// TwinCAT 3 PLC project AssemblyDemo
// ProgramVersion: 3.1.4024.0
// libraries:
//   Tc3_Module, * (Beckhoff Automation GmbH)
//   ZApplication, 1.5.8.2 (Zeugwerk GmbH)
//   ZAux, 1.5.8.2 (Zeugwerk GmbH)
//   ZCore, 1.5.8.2 (Zeugwerk GmbH)
//   ZEquipment, 1.5.8.2 (Zeugwerk GmbH)
//   ZPlatform, 1.5.8.2 (Zeugwerk GmbH)
// project tree:
//   ZApp/App/ ZApp.TcPOU
//   ZApp/App/_DataTypes/ ZAppStep.TcDUT
//   ZApp/App/_States/ ZAppSequenceBoot.TcPOU, ZAppSequenceBootFault.TcPOU, ZAppSequenceRunning.TcPOU
//   ZApp/App/_SubObjects/ ZAppSequence.TcPOU
//   ZApp/Com/_DataTypes/ ZCom.TcDUT, ZComUnit.TcDUT
//   ZApp/Data/_DataTypes/ ZData.TcDUT, ZDataMachine.TcDUT, ZDataConfig.TcDUT, ZDataCalibration.TcDUT, ZDataRecipe.TcDUT
//   ZApp/Unit/Assembly/ AssemblyUnit.TcPOU, AssemblyUnitProgram.TcPOU, IAssembly.TcIO
//   ZApp/Unit/Assembly/_Com/ AssemblyCom.TcDUT, AssemblyComPublish.TcDUT, AssemblyComPublishEquipment.TcDUT, AssemblyComRef.TcDUT, AssemblyComRequest.TcDUT, AssemblyComSubscribe.TcDUT, AssemblyComSubscribeEquipment.TcDUT
//   ZApp/Unit/Assembly/_DataTypes/ ActuatorHorizontalListenerStep.TcDUT, AssemblyState.TcDUT, AssemblyStep.TcDUT
//   ZApp/Unit/Assembly/_Data/ AssemblyDataCalibration.TcDUT, AssemblyDataConfig.TcDUT, AssemblyDataMachine.TcDUT, AssemblyDataRef.TcDUT
//   ZApp/Unit/Assembly/_Equipment/ ActuatorHorizontalListener.TcPOU, AssemblyActuator.TcPOU, AssemblyActuatorGripper.TcPOU, AssemblyActuatorHorizontal.TcPOU, AssemblyAxis.TcPOU, AssemblyEquipment.TcPOU, AssemblyFieldbus.TcPOU, AssemblyIo.TcPOU, AssemblyLinkedUnit.TcPOU, PneumaticsOkActuatorListener.TcPOU
//   ZApp/Unit/Assembly/_States/ AssemblySequenceAutomatic.TcPOU, AssemblySequenceBoot.TcPOU, AssemblySequenceFaultReaction.TcPOU, AssemblySequenceGoHome.TcPOU, AssemblySequenceStop.TcPOU
//   ZApp/Unit/Assembly/_SubObjects/ AssemblyContainer.TcPOU, AssemblySequence.TcPOU
//   ZApp/Unit/Drilling/ DrillingUnit.TcPOU, DrillingUnitProgram.TcPOU, IDrilling.TcIO
//   ZApp/Unit/Drilling/_Com/ DrillingCom.TcDUT, DrillingComPublish.TcDUT, DrillingComPublishEquipment.TcDUT, DrillingComRef.TcDUT, DrillingComRequest.TcDUT, DrillingComSubscribe.TcDUT, DrillingComSubscribeEquipment.TcDUT
//   ZApp/Unit/Drilling/_DataTypes/ DrillingState.TcDUT, DrillingStep.TcDUT
//   ZApp/Unit/Drilling/_Data/ DrillingDataCalibration.TcDUT, DrillingDataConfig.TcDUT, DrillingDataMachine.TcDUT, DrillingDataRef.TcDUT
//   ZApp/Unit/Drilling/_Equipment/ DrillingActuator.TcPOU, DrillingActuatorVertical.TcPOU, DrillingAxis.TcPOU, DrillingEquipment.TcPOU, DrillingFieldbus.TcPOU, DrillingIo.TcPOU, DrillingLinkedUnit.TcPOU
//   ZApp/Unit/Drilling/_States/ DrillingSequenceAutomatic.TcPOU, DrillingSequenceBoot.TcPOU, DrillingSequenceFaultReaction.TcPOU, DrillingSequenceGoHome.TcPOU, DrillingSequenceStop.TcPOU
//   ZApp/Unit/Drilling/_SubObjects/ DrillingContainer.TcPOU, DrillingSequence.TcPOU
//   ZApp/Unit/QualityInspection/ IQualityInspection.TcIO, QualityInspectionUnit.TcPOU, QualityInspectionUnitProgram.TcPOU
//   ZApp/Unit/QualityInspection/_Com/ QualityInspectionCom.TcDUT, QualityInspectionComPublish.TcDUT, QualityInspectionComPublishEquipment.TcDUT, QualityInspectionComRef.TcDUT, QualityInspectionComRequest.TcDUT, QualityInspectionComSubscribe.TcDUT, QualityInspectionComSubscribeEquipment.TcDUT
//   ZApp/Unit/QualityInspection/_DataTypes/ QualityInspectionState.TcDUT, QualityInspectionStep.TcDUT
//   ZApp/Unit/QualityInspection/_Data/ QualityInspectionDataCalibration.TcDUT, QualityInspectionDataConfig.TcDUT, QualityInspectionDataMachine.TcDUT, QualityInspectionDataRef.TcDUT
//   ZApp/Unit/QualityInspection/_Equipment/ QualityInspectionActuator.TcPOU, QualityInspectionAxis.TcPOU, QualityInspectionEquipment.TcPOU, QualityInspectionFieldbus.TcPOU, QualityInspectionIo.TcPOU, QualityInspectionLinkedUnit.TcPOU
//   ZApp/Unit/QualityInspection/_States/ QualityInspectionSequenceAutomatic.TcPOU, QualityInspectionSequenceBoot.TcPOU, QualityInspectionSequenceFaultReaction.TcPOU, QualityInspectionSequenceGoHome.TcPOU, QualityInspectionSequenceStop.TcPOU
//   ZApp/Unit/QualityInspection/_SubObjects/ QualityInspectionContainer.TcPOU, QualityInspectionSequence.TcPOU
//   ZApp/Unit/Transport/ ITransport.TcIO, TransportUnit.TcPOU, TransportUnitProgram.TcPOU
//   ZApp/Unit/Transport/_Com/ TransportCom.TcDUT, TransportComPublish.TcDUT, TransportComPublishEquipment.TcDUT, TransportComRef.TcDUT, TransportComRequest.TcDUT, TransportComSubscribe.TcDUT, TransportComSubscribeEquipment.TcDUT
//   ZApp/Unit/Transport/_DataTypes/ TransportState.TcDUT, TransportStep.TcDUT
//   ZApp/Unit/Transport/_Data/ TransportDataCalibration.TcDUT, TransportDataConfig.TcDUT, TransportDataMachine.TcDUT, TransportDataRef.TcDUT
//   ZApp/Unit/Transport/_Equipment/ TransportActuator.TcPOU, TransportActuatorGripper.TcPOU, TransportAxis.TcPOU, TransportEquipment.TcPOU, TransportFieldbus.TcPOU, TransportIo.TcPOU, TransportLinkedUnit.TcPOU
//   ZApp/Unit/Transport/_States/ TransportSequenceAutomatic.TcPOU, TransportSequenceBoot.TcPOU, TransportSequenceFaultReaction.TcPOU, TransportSequenceGoHome.TcPOU, TransportSequenceStop.TcPOU
//   ZApp/Unit/Transport/_SubObjects/ TransportContainer.TcPOU, TransportSequence.TcPOU
//   ZApp/ ZGlobal.TcGVL, ZModuleProgram.TcPOU, ZModuleTask.TcTTO
// real-time tasks:
//   TASK ZModuleTask: cycle T#10ms, priority 20, ADS port 350

CONFIGURATION AssemblyDemo
    RESOURCE PLC ON TwinCAT3
        TASK ZModuleTask(INTERVAL := T#10ms, PRIORITY := 20);
        PROGRAM ZModuleProgram WITH ZModuleTask : ZModuleProgram;
    END_RESOURCE
END_CONFIGURATION

// ---- ZApp/App/_DataTypes/ZAppStep.TcDUT
{attribute 'qualified_only'}
{attribute 'to_string'}
TYPE ZAppStep :
(
  Undefined := 0
  
  ,BootBegin
  ,BootLoadDefaultData
  ,BootEnd
  ,BootFaultBegin
  ,BootFaultEnd 
  ,RunningBegin
  ,RunningEnd   
);
END_TYPE

// ---- ZApp/Com/_DataTypes/ZCom.TcDUT
TYPE ZCom :
STRUCT
  // module context
  App : ZApplication.ApplicationComPublish;
  Alarming : ZApplication.AlarmingCom;
  Messages : ZApplication.MessagingCom;
  
  // unit context
  Unit : ZComUnit;

END_STRUCT
END_TYPE

// ---- ZApp/Com/_DataTypes/ZComUnit.TcDUT
TYPE ZComUnit :
STRUCT
{region "Transport"}
{IF NOT (defined (Transport_disabled))}
  Transport : TransportCom;
  {attribute 'ZId' := '413070d6-61de-4759-aae5-e3ab76278fe1'}
{END_IF}
{endregion}
{region "Drilling"}
{IF NOT (defined (Drilling_disabled))}
  Drilling : DrillingCom;
  {attribute 'ZId' := 'a0f6f6d1-15cf-44f1-8585-ff8bdaab6c0e'}
{END_IF}
{endregion}
{region "Assembly"}
{IF NOT (defined (Assembly_disabled))}
  Assembly : AssemblyCom;
  {attribute 'ZId' := 'fe48c71e-df5c-4f02-81a6-6f01ddca37c0'}
{END_IF}
{endregion}
{region "QualityInspection"}
{IF NOT (defined (QualityInspection_disabled))}
  QualityInspection : QualityInspectionCom;
  {attribute 'ZId' := 'a1721ee9-e163-4dba-818e-d45d6db51cc5'}
{END_IF}
{endregion}
{attribute '__ZwPlcApplicationComUnitDeclaration__'} // Do not remove this attribute! It is used for code generation.
END_STRUCT
END_TYPE

// ---- ZApp/Data/_DataTypes/ZData.TcDUT
TYPE ZData :
STRUCT
  Config : ZDataConfig;
  Machine : ZDataMachine;
  Calibration : ZDataCalibration;
  Recipe : ZDataRecipe;
END_STRUCT
END_TYPE

// ---- ZApp/Data/_DataTypes/ZDataMachine.TcDUT
TYPE ZDataMachine :
STRUCT
{region "Transport"}
{IF NOT (defined (Transport_disabled))}
  Transport : TransportDataMachine;
  {attribute 'ZId' := '413070d6-61de-4759-aae5-e3ab76278fe1'}
{END_IF}
{endregion}
{region "Drilling"}
{IF NOT (defined (Drilling_disabled))}
  Drilling : DrillingDataMachine;
  {attribute 'ZId' := 'a0f6f6d1-15cf-44f1-8585-ff8bdaab6c0e'}
{END_IF}
{endregion}
{region "Assembly"}
{IF NOT (defined (Assembly_disabled))}
  Assembly : AssemblyDataMachine;
  {attribute 'ZId' := 'fe48c71e-df5c-4f02-81a6-6f01ddca37c0'}
{END_IF}
{endregion}
{region "QualityInspection"}
{IF NOT (defined (QualityInspection_disabled))}
  QualityInspection : QualityInspectionDataMachine;
  {attribute 'ZId' := 'a1721ee9-e163-4dba-818e-d45d6db51cc5'}
{END_IF}
{endregion}
{attribute '__ZwPlcApplicationDataMachineDeclaration__'} // Do not remove this attribute! It is used for code generation.
END_STRUCT
END_TYPE

// ---- ZApp/Data/_DataTypes/ZDataConfig.TcDUT
TYPE ZDataConfig :
STRUCT
{region "Transport"}
{IF NOT (defined (Transport_disabled))}
  Transport : TransportDataConfig;
  {attribute 'ZId' := '413070d6-61de-4759-aae5-e3ab76278fe1'}
{END_IF}
{endregion}
{region "Drilling"}
{IF NOT (defined (Drilling_disabled))}
  Drilling : DrillingDataConfig;
  {attribute 'ZId' := 'a0f6f6d1-15cf-44f1-8585-ff8bdaab6c0e'}
{END_IF}
{endregion}
{region "Assembly"}
{IF NOT (defined (Assembly_disabled))}
  Assembly : AssemblyDataConfig;
  {attribute 'ZId' := 'fe48c71e-df5c-4f02-81a6-6f01ddca37c0'}
{END_IF}
{endregion}
{region "QualityInspection"}
{IF NOT (defined (QualityInspection_disabled))}
  QualityInspection : QualityInspectionDataConfig;
  {attribute 'ZId' := 'a1721ee9-e163-4dba-818e-d45d6db51cc5'}
{END_IF}
{endregion}
{attribute '__ZwPlcApplicationDataConfigDeclaration__'} // Do not remove this attribute! It is used for code generation.
END_STRUCT
END_TYPE

// ---- ZApp/Data/_DataTypes/ZDataCalibration.TcDUT
TYPE ZDataCalibration :
STRUCT
{region "Transport"}
{IF NOT (defined (Transport_disabled))}
  Transport : TransportDataCalibration;
  {attribute 'ZId' := '413070d6-61de-4759-aae5-e3ab76278fe1'}
{END_IF}
{endregion}
{region "Drilling"}
{IF NOT (defined (Drilling_disabled))}
  Drilling : DrillingDataCalibration;
  {attribute 'ZId' := 'a0f6f6d1-15cf-44f1-8585-ff8bdaab6c0e'}
{END_IF}
{endregion}
{region "Assembly"}
{IF NOT (defined (Assembly_disabled))}
  Assembly : AssemblyDataCalibration;
  {attribute 'ZId' := 'fe48c71e-df5c-4f02-81a6-6f01ddca37c0'}
{END_IF}
{endregion}
{region "QualityInspection"}
{IF NOT (defined (QualityInspection_disabled))}
  QualityInspection : QualityInspectionDataCalibration;
  {attribute 'ZId' := 'a1721ee9-e163-4dba-818e-d45d6db51cc5'}
{END_IF}
{endregion}
{attribute '__ZwPlcApplicationDataCalibrationDeclaration__'} // Do not remove this attribute! It is used for code generation.
END_STRUCT
END_TYPE

// ---- ZApp/Data/_DataTypes/ZDataRecipe.TcDUT
TYPE ZDataRecipe :
STRUCT
  RecipeParam1 : LREAL;
  RecipeParam2 : LREAL;
  RecipeParam3 : LREAL;
END_STRUCT
END_TYPE

// ---- ZApp/Unit/Assembly/_Com/AssemblyCom.TcDUT
/// This struct contains variables that
/// * are read from outside (e.g. HMI) to retrieve information about the unit's current state and (temporary) parameters (= `publish`) 
/// * are written from outside (e.g. HMI) to control the unit via ADS (= `subscribe`) 
TYPE AssemblyCom :
STRUCT
  Publish : AssemblyComPublish;
  Subscribe : AssemblyComSubscribe;
END_STRUCT
END_TYPE

// ---- ZApp/Unit/Assembly/_Com/AssemblyComPublish.TcDUT
/// this is the container of informations that the unit wants to share with the world outside of the PLC
/// This struct should only be read from by external applications.
TYPE AssemblyComPublish :
STRUCT
  State : ZApplication.UnitStateMachineState; // state the unit is in
  Request : AssemblyComRequest; // booleans that indictate which action is currently possible to perform with this unit
  Equipment : AssemblyComPublishEquipment;  // structs for equipment objects which are used by the bridges
END_STRUCT
END_TYPE

// ---- ZApp/Unit/Assembly/_Com/AssemblyComPublishEquipment.TcDUT
TYPE AssemblyComPublishEquipment :
STRUCT

{region "Vertical : Axis"}
  Vertical : ZApplication.AxisComPublish;
  {attribute 'ZId' := '59ce020b-a4f8-4d7a-a0dc-8b778ee4fde8'}
{endregion}

{region "Horizontal : ActuatorDigital"}
  Horizontal : ZApplication.ActuatorDigitalComPublish;
  HorizontalToAssembly : ZApplication.DigitalComPublish;
  HorizontalToTransport : ZApplication.DigitalComPublish;
  HorizontalAtAssembly : ZApplication.DigitalComPublish;
  HorizontalAtTransport : ZApplication.DigitalComPublish;
  {attribute 'ZId' := 'bf04a1fd-9e2a-444c-be25-15a99c5011b8'}
{endregion}

{region "YellowLight : Digital"}
  YellowLight : ZApplication.DigitalComPublish;
  {attribute 'ZId' := 'd8b54b94-4c20-4805-9de3-a35aa5023c5d'}
{endregion}

{region "RedLight : Digital"}
  RedLight : ZApplication.DigitalComPublish;
  {attribute 'ZId' := '810dce14-d302-4e94-b60a-e39841040373'}
{endregion}

{region "GreenLight : Digital"}
  GreenLight : ZApplication.DigitalComPublish;
  {attribute 'ZId' := 'f5a46fca-074f-4557-8a14-cee504d2eb08'}
{endregion}

{region "PneumaticsOk : Digital"}
  PneumaticsOk : ZApplication.DigitalComPublish;
  {attribute 'ZId' := 'e461ecc5-0720-4dc8-ad47-eeb7ce01769f'}
{endregion}

{region "Gripper : ActuatorDigital"}
  Gripper : ZApplication.ActuatorDigitalComPublish;
  GripperAuf : ZApplication.DigitalComPublish;
  {attribute 'ZId' := 'd18888e4-9abb-463d-b01d-e5fd8694a677'}
{endregion}

{attribute '__ZwPlcUnitComDeclaration__'} // Do not remove this attribute! It is used for code generation.

END_STRUCT
END_TYPE

// ---- ZApp/Unit/Assembly/_Com/AssemblyComRef.TcDUT
/// container for all communication data types that are used by the unit
TYPE AssemblyComRef :
STRUCT
  Publish : REFERENCE TO AssemblyComPublish; 
  Subscribe : REFERENCE TO AssemblyComSubscribe; 
END_STRUCT
END_TYPE

// ---- ZApp/Unit/Assembly/_Com/AssemblyComRequest.TcDUT
TYPE AssemblyComRequest :
STRUCT
  Start : BOOL;
  Stop : BOOL;
  GoHome : BOOL;
  Halt : BOOL;
END_STRUCT
END_TYPE

// ---- ZApp/Unit/Assembly/_Com/AssemblyComSubscribe.TcDUT
TYPE AssemblyComSubscribe :
STRUCT
  Request : AssemblyComRequest; // contains booleans that are used to start a specific sequence.
  Equipment : AssemblyComSubscribeEquipment;  // structs for equipment objects which are used by the bridges
END_STRUCT
END_TYPE

// ---- ZApp/Unit/Assembly/_Com/AssemblyComSubscribeEquipment.TcDUT
TYPE AssemblyComSubscribeEquipment :
STRUCT

{region "Vertical : Axis"}
  Vertical : ZApplication.AxisComSubscribe;
  {attribute 'ZId' := '59ce020b-a4f8-4d7a-a0dc-8b778ee4fde8'}
{endregion}

{region "Horizontal : ActuatorDigital"}
  Horizontal : ZApplication.ActuatorDigitalComSubscribe;
  HorizontalToAssembly : ZApplication.DigitalComSubscribe;
  HorizontalToTransport : ZApplication.DigitalComSubscribe;
  HorizontalAtAssembly : ZApplication.DigitalComSubscribe;
  HorizontalAtTransport : ZApplication.DigitalComSubscribe;
  {attribute 'ZId' := 'bf04a1fd-9e2a-444c-be25-15a99c5011b8'}
{endregion}

{region "YellowLight : Digital"}
  YellowLight : ZApplication.DigitalComSubscribe;
  {attribute 'ZId' := 'd8b54b94-4c20-4805-9de3-a35aa5023c5d'}
{endregion}

{region "RedLight : Digital"}
  RedLight : ZApplication.DigitalComSubscribe;
  {attribute 'ZId' := '810dce14-d302-4e94-b60a-e39841040373'}
{endregion}

{region "GreenLight : Digital"}
  GreenLight : ZApplication.DigitalComSubscribe;
  {attribute 'ZId' := 'f5a46fca-074f-4557-8a14-cee504d2eb08'}
{endregion}

{region "PneumaticsOk : Digital"}
  PneumaticsOk : ZApplication.DigitalComSubscribe;
  {attribute 'ZId' := 'e461ecc5-0720-4dc8-ad47-eeb7ce01769f'}
{endregion}

{region "Gripper : ActuatorDigital"}
  Gripper : ZApplication.ActuatorDigitalComSubscribe;
  GripperAuf : ZApplication.DigitalComSubscribe;
  {attribute 'ZId' := 'd18888e4-9abb-463d-b01d-e5fd8694a677'}
{endregion}

{attribute '__ZwPlcUnitComDeclaration__'} // Do not remove this attribute! It is used for code generation.

END_STRUCT
END_TYPE

// ---- ZApp/Unit/Assembly/_DataTypes/ActuatorHorizontalListenerStep.TcDUT
{attribute 'qualified_only'}
{attribute 'to_string'}
TYPE ActuatorHorizontalListenerStep :
(
  Undefined := 0
  
  ,PreMoveStepBegin
  ,PreMoveStepStartLightBlinking
  ,PreMoveStepCheckAxisVerticalPosition
  ,PreMoveStepEnd
);
END_TYPE

// ---- ZApp/Unit/Assembly/_DataTypes/AssemblyState.TcDUT
/// This enumeration contains all used defined sequences of a unit.
/// Per default a unit makes use of the states that are contained in (UnitStateDefault)[xref:ZApplication.UnitStateDefault]. However,
/// most of the time a unit need to perform some application depend sequences that can be performed by putting the unit into userdefined states.
/// For instance, a robotic unit could use the state (automatic)[xref:ZApplication.UnitStateDefault] to lift an object from point A to point B,
/// a userdefined state could be used to open and close the robotic-units gripper, respectively
{attribute 'qualified_only'}
TYPE AssemblyState :
(
	UserdefinedState1 := ZApplication.UnitStateMachineState.Last+1
);
END_TYPE

// ---- ZApp/Unit/Assembly/_DataTypes/AssemblyStep.TcDUT
/// This enumeration contains all steps that are used by the various sequences of a unit.
/// Sequences use a subrange (***Begin to ***End) of this enumeration.
{attribute 'qualified_only'}
{attribute 'to_string'}
TYPE AssemblyStep :
(
  Undefined := 0
  
  ,BootBegin
  ,BootSwitchOnPneumaticsOkInSimulation
  ,BootEnd 

  ,StopBegin
  ,StopEnd

  ,AutomaticBegin
  ,AutomaticEnd
  
  ,GoHomeBegin
  ,GoHomeGoToHomePos
  ,GoHomeEnd 
  
  ,FaultReactionBegin
  ,FaultReactionEnd
);
END_TYPE

// ---- ZApp/Unit/Assembly/_Data/AssemblyDataCalibration.TcDUT
/// calibration that is determined by calibration sequences of the unit (static offsets, shifts)
TYPE AssemblyDataCalibration :
STRUCT
END_STRUCT
END_TYPE

// ---- ZApp/Unit/Assembly/_Data/AssemblyDataConfig.TcDUT
/// configuration data that is used during boot to configure the Units equipment
TYPE AssemblyDataConfig :
STRUCT
  Simulated : BOOL;
END_STRUCT
END_TYPE

// ---- ZApp/Unit/Assembly/_Data/AssemblyDataMachine.TcDUT
/// machine data that is used through most sequences of the unit (motor speed, axes positions, ...)
TYPE AssemblyDataMachine :
STRUCT
  Slowspeed : LREAL;
  Highspeed : LREAL;
END_STRUCT
END_TYPE

// ---- ZApp/Unit/Assembly/_Data/AssemblyDataRef.TcDUT
/// container for all data that are used by the unit
TYPE AssemblyDataRef :
STRUCT
  Config : REFERENCE TO AssemblyDataConfig; // data required for booting the unit (axes configuration, simulation, parameters that have to be written in PREOP, ...)
  Machine : REFERENCE TO AssemblyDataMachine; // speeds, positions, ...
  Calibration : REFERENCE TO AssemblyDataCalibration; // offsets, shifts of nominal to actual values
END_STRUCT
END_TYPE

// ---- ZApp/Unit/Drilling/_Com/DrillingCom.TcDUT
/// This struct contains variables that
/// * are read from outside (e.g. HMI) to retrieve information about the unit's current state and (temporary) parameters (= `publish`) 
/// * are written from outside (e.g. HMI) to control the unit via ADS (= `subscribe`) 
TYPE DrillingCom :
STRUCT
  Publish : DrillingComPublish;
  Subscribe : DrillingComSubscribe;
END_STRUCT
END_TYPE

// ---- ZApp/Unit/Drilling/_Com/DrillingComPublish.TcDUT
/// this is the container of informations that the unit wants to share with the world outside of the PLC
/// This struct should only be read from by external applications.
TYPE DrillingComPublish :
STRUCT
  State : ZApplication.UnitStateMachineState; // state the unit is in
  Request : DrillingComRequest; // booleans that indictate which action is currently possible to perform with this unit
  Equipment : DrillingComPublishEquipment;  // structs for equipment objects which are used by the bridges
END_STRUCT
END_TYPE

// ---- ZApp/Unit/Drilling/_Com/DrillingComPublishEquipment.TcDUT
TYPE DrillingComPublishEquipment :
STRUCT

{region "Vertical : ActuatorDigital"}
  Vertical : ZApplication.ActuatorDigitalComPublish;
  VerticalZu : ZApplication.DigitalComPublish;
  VerticalAuf : ZApplication.DigitalComPublish;
  VerticalGeschlossen : ZApplication.DigitalComPublish;
  VerticalOffen : ZApplication.DigitalComPublish;
  {attribute 'ZId' := '6edc2aeb-8e0c-4ef7-9533-2d3679311649'}
{endregion}

{attribute '__ZwPlcUnitComDeclaration__'} // Do not remove this attribute! It is used for code generation.

END_STRUCT
END_TYPE

// ---- ZApp/Unit/Drilling/_Com/DrillingComRef.TcDUT
/// container for all communication data types that are used by the unit
TYPE DrillingComRef :
STRUCT
  Publish : REFERENCE TO DrillingComPublish; 
  Subscribe : REFERENCE TO DrillingComSubscribe; 
END_STRUCT
END_TYPE

// ---- ZApp/Unit/Drilling/_Com/DrillingComRequest.TcDUT
TYPE DrillingComRequest :
STRUCT
  Start : BOOL;
  Stop : BOOL;
  GoHome : BOOL;
  Halt : BOOL;
END_STRUCT
END_TYPE

// ---- ZApp/Unit/Drilling/_Com/DrillingComSubscribe.TcDUT
TYPE DrillingComSubscribe :
STRUCT
  Request : DrillingComRequest; // contains booleans that are used to start a specific sequence.
  Equipment : DrillingComSubscribeEquipment;  // structs for equipment objects which are used by the bridges
END_STRUCT
END_TYPE

// ---- ZApp/Unit/Drilling/_Com/DrillingComSubscribeEquipment.TcDUT
TYPE DrillingComSubscribeEquipment :
STRUCT

{region "Vertical : ActuatorDigital"}
  Vertical : ZApplication.ActuatorDigitalComSubscribe;
  VerticalZu : ZApplication.DigitalComSubscribe;
  VerticalAuf : ZApplication.DigitalComSubscribe;
  VerticalGeschlossen : ZApplication.DigitalComSubscribe;
  VerticalOffen : ZApplication.DigitalComSubscribe;
  {attribute 'ZId' := '6edc2aeb-8e0c-4ef7-9533-2d3679311649'}
{endregion}

{attribute '__ZwPlcUnitComDeclaration__'} // Do not remove this attribute! It is used for code generation.

END_STRUCT
END_TYPE

// ---- ZApp/Unit/Drilling/_DataTypes/DrillingState.TcDUT
/// This enumeration contains all used defined sequences of a unit.
/// Per default a unit makes use of the states that are contained in (UnitStateDefault)[xref:ZApplication.UnitStateDefault]. However,
/// most of the time a unit need to perform some application depend sequences that can be performed by putting the unit into userdefined states.
/// For instance, a robotic unit could use the state (automatic)[xref:ZApplication.UnitStateDefault] to lift an object from point A to point B,
/// a userdefined state could be used to open and close the robotic-units gripper, respectively
{attribute 'qualified_only'}
TYPE DrillingState :
(
	UserdefinedState1 := ZApplication.UnitStateMachineState.Last+1
);
END_TYPE

// ---- ZApp/Unit/Drilling/_DataTypes/DrillingStep.TcDUT
/// This enumeration contains all steps that are used by the various sequences of a unit.
/// Sequences use a subrange (***Begin to ***End) of this enumeration.
{attribute 'qualified_only'}
{attribute 'to_string'}
TYPE DrillingStep :
(
  Undefined := 0
  
  ,BootBegin
  ,BootEnd 

  ,StopBegin
  ,StopEnd

  ,AutomaticBegin
  ,AutomaticEnd
  
  ,GoHomeBegin
  ,GoHomeEnd 
  
  ,FaultReactionBegin
  ,FaultReactionEnd
);
END_TYPE

// ---- ZApp/Unit/Drilling/_Data/DrillingDataCalibration.TcDUT
/// calibration that is determined by calibration sequences of the unit (static offsets, shifts)
TYPE DrillingDataCalibration :
STRUCT
END_STRUCT
END_TYPE

// ---- ZApp/Unit/Drilling/_Data/DrillingDataConfig.TcDUT
/// configuration data that is used during boot to configure the Units equipment
TYPE DrillingDataConfig :
STRUCT
  Simulated : BOOL;
END_STRUCT
END_TYPE

// ---- ZApp/Unit/Drilling/_Data/DrillingDataMachine.TcDUT
/// machine data that is used through most sequences of the unit (motor speed, axes positions, ...)
TYPE DrillingDataMachine :
STRUCT
  Slowspeed : LREAL;
  Highspeed : LREAL;
END_STRUCT
END_TYPE

// ---- ZApp/Unit/Drilling/_Data/DrillingDataRef.TcDUT
/// container for all data that are used by the unit
TYPE DrillingDataRef :
STRUCT
  Config : REFERENCE TO DrillingDataConfig; // data required for booting the unit (axes configuration, simulation, parameters that have to be written in PREOP, ...)
  Machine : REFERENCE TO DrillingDataMachine; // speeds, positions, ...
  Calibration : REFERENCE TO DrillingDataCalibration; // offsets, shifts of nominal to actual values
END_STRUCT
END_TYPE

// ---- ZApp/Unit/QualityInspection/_Com/QualityInspectionCom.TcDUT
/// This struct contains variables that
/// * are read from outside (e.g. HMI) to retrieve information about the unit's current state and (temporary) parameters (= `publish`) 
/// * are written from outside (e.g. HMI) to control the unit via ADS (= `subscribe`) 
TYPE QualityInspectionCom :
STRUCT
  Publish : QualityInspectionComPublish;
  Subscribe : QualityInspectionComSubscribe;
END_STRUCT
END_TYPE

// ---- ZApp/Unit/QualityInspection/_Com/QualityInspectionComPublish.TcDUT
/// this is the container of informations that the unit wants to share with the world outside of the PLC
/// This struct should only be read from by external applications.
TYPE QualityInspectionComPublish :
STRUCT
  State : ZApplication.UnitStateMachineState; // state the unit is in
  Request : QualityInspectionComRequest; // booleans that indictate which action is currently possible to perform with this unit
  Equipment : QualityInspectionComPublishEquipment;  // structs for equipment objects which are used by the bridges
END_STRUCT
END_TYPE

// ---- ZApp/Unit/QualityInspection/_Com/QualityInspectionComPublishEquipment.TcDUT
TYPE QualityInspectionComPublishEquipment :
STRUCT

{region "TriggerCam : PulsedOutput"}
  TriggerCam : ZApplication.ImpulseOutputComPublish;
  {attribute 'ZId' := 'c63d51c9-4589-40b4-ac78-45c3ff2f3b57'}
{endregion}

{region "EnableLight : Digital"}
  EnableLight : ZApplication.DigitalComPublish;
  {attribute 'ZId' := '57b0de1b-3452-4c6c-9481-eeca6b7d3a02'}
{endregion}

{region "CamOk : Digital"}
  CamOk : ZApplication.DigitalComPublish;
  {attribute 'ZId' := '27a646f9-ab74-4898-af0f-5400552173e7'}
{endregion}

{attribute '__ZwPlcUnitComDeclaration__'} // Do not remove this attribute! It is used for code generation.

END_STRUCT
END_TYPE

// ---- ZApp/Unit/QualityInspection/_Com/QualityInspectionComRef.TcDUT
/// container for all communication data types that are used by the unit
TYPE QualityInspectionComRef :
STRUCT
  Publish : REFERENCE TO QualityInspectionComPublish; 
  Subscribe : REFERENCE TO QualityInspectionComSubscribe; 
END_STRUCT
END_TYPE

// ---- ZApp/Unit/QualityInspection/_Com/QualityInspectionComRequest.TcDUT
TYPE QualityInspectionComRequest :
STRUCT
  Start : BOOL;
  Stop : BOOL;
  GoHome : BOOL;
  Halt : BOOL;
END_STRUCT
END_TYPE

// ---- ZApp/Unit/QualityInspection/_Com/QualityInspectionComSubscribe.TcDUT
TYPE QualityInspectionComSubscribe :
STRUCT
  Request : QualityInspectionComRequest; // contains booleans that are used to start a specific sequence.
  Equipment : QualityInspectionComSubscribeEquipment;  // structs for equipment objects which are used by the bridges
END_STRUCT
END_TYPE

// ---- ZApp/Unit/QualityInspection/_Com/QualityInspectionComSubscribeEquipment.TcDUT
TYPE QualityInspectionComSubscribeEquipment :
STRUCT

{region "TriggerCam : PulsedOutput"}
  TriggerCam : ZApplication.ImpulseOutputComSubscribe;
  {attribute 'ZId' := 'c63d51c9-4589-40b4-ac78-45c3ff2f3b57'}
{endregion}

{region "EnableLight : Digital"}
  EnableLight : ZApplication.DigitalComSubscribe;
  {attribute 'ZId' := '57b0de1b-3452-4c6c-9481-eeca6b7d3a02'}
{endregion}

{region "CamOk : Digital"}
  CamOk : ZApplication.DigitalComSubscribe;
  {attribute 'ZId' := '27a646f9-ab74-4898-af0f-5400552173e7'}
{endregion}

{attribute '__ZwPlcUnitComDeclaration__'} // Do not remove this attribute! It is used for code generation.

END_STRUCT
END_TYPE

// ---- ZApp/Unit/QualityInspection/_DataTypes/QualityInspectionState.TcDUT
/// This enumeration contains all used defined sequences of a unit.
/// Per default a unit makes use of the states that are contained in (UnitStateDefault)[xref:ZApplication.UnitStateDefault]. However,
/// most of the time a unit need to perform some application depend sequences that can be performed by putting the unit into userdefined states.
/// For instance, a robotic unit could use the state (automatic)[xref:ZApplication.UnitStateDefault] to lift an object from point A to point B,
/// a userdefined state could be used to open and close the robotic-units gripper, respectively
{attribute 'qualified_only'}
TYPE QualityInspectionState :
(
	UserdefinedState1 := ZApplication.UnitStateMachineState.Last+1
);
END_TYPE

// ---- ZApp/Unit/QualityInspection/_DataTypes/QualityInspectionStep.TcDUT
/// This enumeration contains all steps that are used by the various sequences of a unit.
/// Sequences use a subrange (***Begin to ***End) of this enumeration.
{attribute 'qualified_only'}
{attribute 'to_string'}
TYPE QualityInspectionStep :
(
  Undefined := 0
  
  ,BootBegin
  ,BootEnd 

  ,StopBegin
  ,StopEnd

  ,AutomaticBegin
  ,AutomaticEnableLight
  ,AutomaticTriggerCam
  ,AutomaticWaitTillCamSendsOk
  ,AutomaticEnd
  
  ,GoHomeBegin
  ,GoHomeEnd 
  
  ,FaultReactionBegin
  ,FaultReactionEnd
);
END_TYPE

// ---- ZApp/Unit/QualityInspection/_Data/QualityInspectionDataCalibration.TcDUT
/// calibration that is determined by calibration sequences of the unit (static offsets, shifts)
TYPE QualityInspectionDataCalibration :
STRUCT
END_STRUCT
END_TYPE

// ---- ZApp/Unit/QualityInspection/_Data/QualityInspectionDataConfig.TcDUT
/// configuration data that is used during boot to configure the Units equipment
TYPE QualityInspectionDataConfig :
STRUCT
  Simulated : BOOL;
END_STRUCT
END_TYPE

// ---- ZApp/Unit/QualityInspection/_Data/QualityInspectionDataMachine.TcDUT
/// machine data that is used through most sequences of the unit (motor speed, axes positions, ...)
TYPE QualityInspectionDataMachine :
STRUCT
  Slowspeed : LREAL;
  Highspeed : LREAL;
END_STRUCT
END_TYPE

// ---- ZApp/Unit/QualityInspection/_Data/QualityInspectionDataRef.TcDUT
/// container for all data that are used by the unit
TYPE QualityInspectionDataRef :
STRUCT
  Config : REFERENCE TO QualityInspectionDataConfig; // data required for booting the unit (axes configuration, simulation, parameters that have to be written in PREOP, ...)
  Machine : REFERENCE TO QualityInspectionDataMachine; // speeds, positions, ...
  Calibration : REFERENCE TO QualityInspectionDataCalibration; // offsets, shifts of nominal to actual values
END_STRUCT
END_TYPE

// ---- ZApp/Unit/Transport/_Com/TransportCom.TcDUT
/// This struct contains variables that
/// * are read from outside (e.g. HMI) to retrieve information about the unit's current state and (temporary) parameters (= `publish`) 
/// * are written from outside (e.g. HMI) to control the unit via ADS (= `subscribe`) 
TYPE TransportCom :
STRUCT
  Publish : TransportComPublish;
  Subscribe : TransportComSubscribe;
END_STRUCT
END_TYPE

// ---- ZApp/Unit/Transport/_Com/TransportComPublish.TcDUT
/// this is the container of informations that the unit wants to share with the world outside of the PLC
/// This struct should only be read from by external applications.
TYPE TransportComPublish :
STRUCT
  State : ZApplication.UnitStateMachineState; // state the unit is in
  Request : TransportComRequest; // booleans that indictate which action is currently possible to perform with this unit
  Equipment : TransportComPublishEquipment;  // structs for equipment objects which are used by the bridges
END_STRUCT
END_TYPE

// ---- ZApp/Unit/Transport/_Com/TransportComPublishEquipment.TcDUT
TYPE TransportComPublishEquipment :
STRUCT

{region "HorizontalX : Axis"}
  HorizontalX : ZApplication.AxisComPublish;
  {attribute 'ZId' := 'b48886d3-effd-43af-8c1e-4c35e310bf5b'}
{endregion}

{region "VerticalZ : Axis"}
  VerticalZ : ZApplication.AxisComPublish;
  {attribute 'ZId' := '82c3e667-8dc4-4ea4-a1fc-9c83583bfea0'}
{endregion}

{region "Gripper : ActuatorDigital"}
  Gripper : ZApplication.ActuatorDigitalComPublish;
  GripperClose : ZApplication.DigitalComPublish;
  GripperOpen : ZApplication.DigitalComPublish;
  GripperIsClosed : ZApplication.DigitalComPublish;
  GripperIsOpen : ZApplication.DigitalComPublish;
  {attribute 'ZId' := '5d1fe583-4573-4e37-9380-49c474c02543'}
{endregion}

{attribute '__ZwPlcUnitComDeclaration__'} // Do not remove this attribute! It is used for code generation.

END_STRUCT
END_TYPE

// ---- ZApp/Unit/Transport/_Com/TransportComRef.TcDUT
/// container for all communication data types that are used by the unit
TYPE TransportComRef :
STRUCT
  Publish : REFERENCE TO TransportComPublish; 
  Subscribe : REFERENCE TO TransportComSubscribe; 
END_STRUCT
END_TYPE

// ---- ZApp/Unit/Transport/_Com/TransportComRequest.TcDUT
TYPE TransportComRequest :
STRUCT
  Start : BOOL;
  Stop : BOOL;
  GoHome : BOOL;
  Halt : BOOL;
END_STRUCT
END_TYPE

// ---- ZApp/Unit/Transport/_Com/TransportComSubscribe.TcDUT
TYPE TransportComSubscribe :
STRUCT
  Request : TransportComRequest; // contains booleans that are used to start a specific sequence.
  Equipment : TransportComSubscribeEquipment;  // structs for equipment objects which are used by the bridges
END_STRUCT
END_TYPE

// ---- ZApp/Unit/Transport/_Com/TransportComSubscribeEquipment.TcDUT
TYPE TransportComSubscribeEquipment :
STRUCT

{region "HorizontalX : Axis"}
  HorizontalX : ZApplication.AxisComSubscribe;
  {attribute 'ZId' := 'b48886d3-effd-43af-8c1e-4c35e310bf5b'}
{endregion}

{region "VerticalZ : Axis"}
  VerticalZ : ZApplication.AxisComSubscribe;
  {attribute 'ZId' := '82c3e667-8dc4-4ea4-a1fc-9c83583bfea0'}
{endregion}

{region "Gripper : ActuatorDigital"}
  Gripper : ZApplication.ActuatorDigitalComSubscribe;
  GripperClose : ZApplication.DigitalComSubscribe;
  GripperOpen : ZApplication.DigitalComSubscribe;
  GripperIsClosed : ZApplication.DigitalComSubscribe;
  GripperIsOpen : ZApplication.DigitalComSubscribe;
  {attribute 'ZId' := '5d1fe583-4573-4e37-9380-49c474c02543'}
{endregion}

{attribute '__ZwPlcUnitComDeclaration__'} // Do not remove this attribute! It is used for code generation.

END_STRUCT
END_TYPE

// ---- ZApp/Unit/Transport/_DataTypes/TransportState.TcDUT
/// This enumeration contains all used defined sequences of a unit.
/// Per default a unit makes use of the states that are contained in (UnitStateDefault)[xref:ZApplication.UnitStateDefault]. However,
/// most of the time a unit need to perform some application depend sequences that can be performed by putting the unit into userdefined states.
/// For instance, a robotic unit could use the state (automatic)[xref:ZApplication.UnitStateDefault] to lift an object from point A to point B,
/// a userdefined state could be used to open and close the robotic-units gripper, respectively
{attribute 'qualified_only'}
TYPE TransportState :
(
	UserdefinedState1 := ZApplication.UnitStateMachineState.Last+1
);
END_TYPE

// ---- ZApp/Unit/Transport/_DataTypes/TransportStep.TcDUT
/// This enumeration contains all steps that are used by the various sequences of a unit.
/// Sequences use a subrange (***Begin to ***End) of this enumeration.
{attribute 'qualified_only'}
{attribute 'to_string'}
TYPE TransportStep :
(
  Undefined := 0
  
  ,BootBegin
  ,BootEnd 

  ,StopBegin
  ,StopEnd

  ,AutomaticBegin
  ,AutomaticInitializeMovements  
  ,AutomaticMoveToLeftPos
  ,AutomaticWaitSomeTime
  ,AutomaticMoveVerticalDown
  ,AutomaticCloseGripper
  ,AutomaticMoveVerticalToTopPos  
  ,AutomaticWaitSomeMoreTime
  ,AutomaticMoveToRightPos
  ,AutomaticCleanUp
  ,AutomaticOpenGripper
  ,AutomaticMoveToCamPos
  ,AutomaticStartQualityInspection
  ,AutomaticEnd
  
  ,GoHomeBegin
  ,GoHomeStartHomingOfChilds
  ,GoHomeVerticalUp
  ,GoHomeHorizontalToRightPos
  ,GoHomeUnlockQualityInspection
  ,GoHomeEnd 
  
  ,FaultReactionBegin
  ,FaultReactionVerticalUp
  ,FaultReactionEnd
);
END_TYPE

// ---- ZApp/Unit/Transport/_Data/TransportDataCalibration.TcDUT
/// calibration that is determined by calibration sequences of the unit (static offsets, shifts)
TYPE TransportDataCalibration :
STRUCT
END_STRUCT
END_TYPE

// ---- ZApp/Unit/Transport/_Data/TransportDataConfig.TcDUT
/// configuration data that is used during boot to configure the Units equipment
TYPE TransportDataConfig :
STRUCT
  Simulated : BOOL;
END_STRUCT
END_TYPE

// ---- ZApp/Unit/Transport/_Data/TransportDataMachine.TcDUT
/// machine data that is used through most sequences of the unit (motor speed, axes positions, ...)
TYPE TransportDataMachine :
STRUCT
  Slowspeed : LREAL;
  Highspeed : LREAL;
  
  HorizontalLeftPos : LREAL;
  HorizontalRightPos : LREAL;
  HorizontalCamPos : LREAL;
  HorizontalHomePos : LREAL;
  
  VerticalTopPos : LREAL;
  VerticalBottomPos : LREAL;
  VerticalHomePos : LREAL;
END_STRUCT
END_TYPE

// ---- ZApp/Unit/Transport/_Data/TransportDataRef.TcDUT
/// container for all data that are used by the unit
TYPE TransportDataRef :
STRUCT
  Config : REFERENCE TO TransportDataConfig; // data required for booting the unit (axes configuration, simulation, parameters that have to be written in PREOP, ...)
  Machine : REFERENCE TO TransportDataMachine; // speeds, positions, ...
  Calibration : REFERENCE TO TransportDataCalibration; // offsets, shifts of nominal to actual values
END_STRUCT
END_TYPE

// ---- ZApp/ZGlobal.TcGVL
{attribute 'qualified_only'}
VAR_GLOBAL
  Com : ZCom;
END_VAR
VAR_GLOBAL PERSISTENT
  Data : ZData;
END_VAR

// ---- ZApp/Unit/Assembly/IAssembly.TcIO
INTERFACE IAssembly EXTENDS ZApplication.IUnit

END_INTERFACE

// ---- ZApp/Unit/Drilling/IDrilling.TcIO
INTERFACE IDrilling EXTENDS ZApplication.IUnit

END_INTERFACE

// ---- ZApp/Unit/QualityInspection/IQualityInspection.TcIO
INTERFACE IQualityInspection EXTENDS ZApplication.IUnit

END_INTERFACE

// ---- ZApp/Unit/Transport/ITransport.TcIO
INTERFACE ITransport EXTENDS ZApplication.IUnit

END_INTERFACE

// ---- ZApp/ZModuleProgram.TcPOU
/// Zeugwerk Application
PROGRAM ZModuleProgram
VAR_INPUT
{region "ZModuleProgram : Utility"}
  App : ZApp(name:='Zeugwerk-Application Template', com:=ZGlobal.Com.App);
  Datetime : ZAux.DateTimeUM;
  {attribute 'ZId' := ''}
{endregion}
{region "ZModuleProgram : Logging"}
  Alarming : ZApplication.Alarming(App, datetime := Datetime, com := ZGlobal.Com.Alarming);
  LoggerHmi : ZApplication.Messaging(App, datetime := Datetime, com := ZGlobal.Com.Messages);
  LoggerFile : ZAux.LoggerFile7FF(App, datetime := Datetime, filePath:='C:\Zeugwerk\logs\messages.log', target:='');
  Logger : ZAux.Logging;
  {attribute 'ZId' := ''}
{endregion}  
{attribute '__ZwPlcApplicationModuleProgramDeclaration__'} // Do not remove this attribute! It is used for code generation.
{region "Transport"}
{undefine RunInSeparateProgram}
{IF NOT (defined (Transport_disabled)) AND NOT (defined (RunInSeparateProgram))}
  Transport : TransportUnit(name := 'Transport', // name of the unit (for logging)
					  parent := App, // caller of the Unit's cyclic method. If the Unit runs in its own context use 0
						configdata := ZGlobal.Data.Config.Transport,
						machinedata := ZGlobal.Data.Machine.Transport,
						calibrationdata := ZGlobal.Data.Calibration.Transport,
						com := ZGlobal.Com.Unit.Transport);
  {attribute 'section' := '__ZwPlcUnitProgramDeclaration__'}
  {attribute 'ZId' := '413070d6-61de-4759-aae5-e3ab76278fe1'}
{END_IF}
{endregion}
{region "Drilling"}
{undefine RunInSeparateProgram}
{IF NOT (defined (Drilling_disabled)) AND NOT (defined (RunInSeparateProgram))}
  Drilling : DrillingUnit(name := 'Drilling', // name of the unit (for logging)
					  parent := App, // caller of the Unit's cyclic method. If the Unit runs in its own context use 0
						configdata := ZGlobal.Data.Config.Drilling,
						machinedata := ZGlobal.Data.Machine.Drilling,
						calibrationdata := ZGlobal.Data.Calibration.Drilling,
						com := ZGlobal.Com.Unit.Drilling);
  {attribute 'section' := '__ZwPlcUnitProgramDeclaration__'}
  {attribute 'ZId' := 'a0f6f6d1-15cf-44f1-8585-ff8bdaab6c0e'}
{END_IF}
{endregion}
{region "Assembly"}
{undefine RunInSeparateProgram}
{IF NOT (defined (Assembly_disabled)) AND NOT (defined (RunInSeparateProgram))}
  Assembly : AssemblyUnit(name := 'Assembly', // name of the unit (for logging)
					  parent := App, // caller of the Unit's cyclic method. If the Unit runs in its own context use 0
						configdata := ZGlobal.Data.Config.Assembly,
						machinedata := ZGlobal.Data.Machine.Assembly,
						calibrationdata := ZGlobal.Data.Calibration.Assembly,
						com := ZGlobal.Com.Unit.Assembly);
  {attribute 'section' := '__ZwPlcUnitProgramDeclaration__'}
  {attribute 'ZId' := 'fe48c71e-df5c-4f02-81a6-6f01ddca37c0'}
{END_IF}
{endregion}
{region "QualityInspection"}
{undefine RunInSeparateProgram}
{IF NOT (defined (QualityInspection_disabled)) AND NOT (defined (RunInSeparateProgram))}
  QualityInspection : QualityInspectionUnit(name := 'QualityInspection', // name of the unit (for logging)
					  parent := App, // caller of the Unit's cyclic method. If the Unit runs in its own context use 0
						configdata := ZGlobal.Data.Config.QualityInspection,
						machinedata := ZGlobal.Data.Machine.QualityInspection,
						calibrationdata := ZGlobal.Data.Calibration.QualityInspection,
						com := ZGlobal.Com.Unit.QualityInspection);
  {attribute 'section' := '__ZwPlcUnitProgramDeclaration__'}
  {attribute 'ZId' := 'a1721ee9-e163-4dba-818e-d45d6db51cc5'}
{END_IF}
{endregion}
{attribute '__ZwPlcUnitProgramDeclaration__'} // Do not remove this attribute! It is used for code generation.
END_VAR

{region "ZModuleProgram : Utility"}
  Datetime.Cyclic();
  App.Cyclic();
  {attribute 'ZId' := ''}
{endregion}
{attribute '__ZwPlcApplicationModuleProgramImplementation__'} // Do not remove this attribute! It is used for code generation.

METHOD SetLoggerLevel
VAR_INPUT
  level : ZCore.LogLevel;
END_VAR
LoggerFile.MinimumLevel := level;
END_METHOD

END_PROGRAM

// ---- ZApp/App/ZApp.TcPOU
FUNCTION_BLOCK ZApp EXTENDS ZApplication.Application
VAR
  _boot : ZAppSequenceBoot;
  _bootFault : ZAppSequenceBootFault;
  _running : ZAppSequenceRunning;
END_VAR

METHOD FB_init : BOOL
VAR_INPUT
  bInitRetains : BOOL; /// if TRUE, the retain variables are initialized (warm start / cold start)
  bInCopyCode : BOOL; /// if TRUE, the instance afterwards gets moved into the copy code (online change)
  name : ZCore.ZString;
  com : REFERENCE TO ZApplication.ApplicationComPublish;
END_VAR
SetBootSequence(_boot);
SetBootFaultSequence(_bootFault);
SetRunningSequence(_running);
END_METHOD

END_FUNCTION_BLOCK

// ---- ZApp/App/_States/ZAppSequenceBoot.TcPOU
FUNCTION_BLOCK ZAppSequenceBoot EXTENDS ZAppSequence IMPLEMENTS ZCore.ISequence
VAR
  _step : ZCore.Step(ZAppStep.BootBegin, ZAppStep.BootEnd);
END_VAR

IF OnStart(_step)
THEN
  // init custom sequence variables here ...
END_IF

REPEAT
  LogStep();

  CASE _step.Index OF
    (* -------------------------------------------------------------------------------------------------------------------------------- *)
    ZAppStep.BootBegin:
    (* -------------------------------------------------------------------------------------------------------------------------------- *)
    
      IF _step.OnEntry()
      THEN
        ZModuleProgram.SetLoggerLevel(ZCore.LogLevel.Trace);
        ZModuleProgram.Logger.AddLogger(ZModuleProgram.LoggerFile);        
        {attribute '__ZwPlcAppZComModuleContext__'} // Do not remove this attribute! It is used for code generation.      
      END_IF
      
	  IF ZModuleProgram.Datetime.State <> ZCore.ObjectState.Booting
      THEN
        _step.SetNext(ZAppStep.BootLoadDefaultData);        
      END_IF
      
    (* -------------------------------------------------------------------------------------------------------------------------------- *)
    ZAppStep.BootLoadDefaultData:
    (* -------------------------------------------------------------------------------------------------------------------------------- *)

      {warning 'The application is loading the default config data on every restart!'}
      LoadDefaultConfigData();
      
      IF IsCommissioning()
      THEN
        LoadDefaultData();
      END_IF
      
      _step.SetNext(ZAppStep.BootEnd);
      
    (* -------------------------------------------------------------------------------------------------------------------------------- *)
    ZAppStep.BootEnd:
    (* -------------------------------------------------------------------------------------------------------------------------------- *)
      SetBusy(FALSE);
      
  ELSE
    Abort('sequence contains unhandled step');
  END_CASE
UNTIL _step.IsNotRepeatable() OR_ELSE NOT Busy END_REPEAT

METHOD  IsCommissioning : BOOL
IsCommissioning := TRUE;
END_METHOD

METHOD FINAL LoadDefaultConfigData

{region "Transport"}
  {IF NOT (defined (Transport_disabled))}
  ZGlobal.Data.Config.Transport.Simulated := TRUE;
  {region "UserInitCode"}
  // put your individual init code for this unit here
  ZGlobal.Data.Machine.Transport.Highspeed := 10.0;
  ZGlobal.Data.Machine.Transport.Slowspeed := 2.0;
        
  ZGlobal.Data.Machine.Transport.HorizontalLeftPos := 2.0;
  ZGlobal.Data.Machine.Transport.HorizontalRightPos := 8.0;
  ZGlobal.Data.Machine.Transport.HorizontalHomePos := 0.0;
        
  ZGlobal.Data.Machine.Transport.VerticalBottomPos := 5.0;
  ZGlobal.Data.Machine.Transport.VerticalTopPos := 2.0;
  ZGlobal.Data.Machine.Transport.VerticalHomePos := 0.0;
  {endregion}
  {END_IF}
  {attribute 'ZId' := '413070d6-61de-4759-aae5-e3ab76278fe1'}
{endregion}

{region "Drilling"}
  {IF NOT (defined (Drilling_disabled))}
  ZGlobal.Data.Config.Drilling.Simulated := TRUE;
  {region "UserInitCode"}
  // put your individual init code for this unit here
  {endregion}
  {END_IF}
  {attribute 'ZId' := 'a0f6f6d1-15cf-44f1-8585-ff8bdaab6c0e'}
{endregion}

{region "Assembly"}
  {IF NOT (defined (Assembly_disabled))}
  ZGlobal.Data.Config.Assembly.Simulated := TRUE;
  {region "UserInitCode"}
  // put your individual init code for this unit here
  {endregion}
  {END_IF}
  {attribute 'ZId' := 'fe48c71e-df5c-4f02-81a6-6f01ddca37c0'}
{endregion}

{region "QualityInspection"}
  {IF NOT (defined (QualityInspection_disabled))}
  ZGlobal.Data.Config.QualityInspection.Simulated := TRUE;
  {region "UserInitCode"}
  // put your individual init code for this unit here
  {endregion}
  {END_IF}
  {attribute 'ZId' := 'a1721ee9-e163-4dba-818e-d45d6db51cc5'}
{endregion}

{attribute '__ZwPlcUnitLoadDefaultConfigData__'} // Do not remove this attribute! It is used for code generation.
END_METHOD

METHOD FINAL LoadDefaultData

{attribute '__ZwPlcUnitLoadDefaultData__'} // Do not remove this attribute! It is used for code generation.
END_METHOD

END_FUNCTION_BLOCK

// ---- ZApp/App/_SubObjects/ZAppSequence.TcPOU
FUNCTION_BLOCK ABSTRACT ZAppSequence EXTENDS ZApplication.Sequence IMPLEMENTS ZCore.ISequence

METHOD StepDecoded : ZCore.ZString
VAR_INPUT
  stepIndex : INT;
END_VAR
VAR_INST
  _stepIndexDecoded : ZAppStep;
END_VAR
_stepIndexDecoded := stepIndex;
StepDecoded := TO_STRING(_stepIndexDecoded);
END_METHOD

END_FUNCTION_BLOCK

// ---- ZApp/App/_States/ZAppSequenceBootFault.TcPOU
FUNCTION_BLOCK ZAppSequenceBootFault EXTENDS ZAppSequence IMPLEMENTS ZCore.ISequence
VAR
  _step : ZCore.Step(ZAppStep.BootFaultBegin, ZAppStep.BootFaultEnd);
END_VAR

IF OnStart(_step)
THEN
  // init custom sequence variables here ...
END_IF

REPEAT
  LogStep();

  CASE _step.Index OF
    (* -------------------------------------------------------------------------------------------------------------------------------- *)
    ZAppStep.BootFaultBegin:
    (* -------------------------------------------------------------------------------------------------------------------------------- *)
      _step.SetNext(ZAppStep.BootFaultEnd);
      
    (* -------------------------------------------------------------------------------------------------------------------------------- *)
    ZAppStep.BootFaultEnd:
    (* -------------------------------------------------------------------------------------------------------------------------------- *)
      SetBusy(FALSE);
      
  ELSE
    Abort('sequence contains unhandled step');
  END_CASE
UNTIL _step.IsNotRepeatable() OR_ELSE NOT Busy END_REPEAT

END_FUNCTION_BLOCK

// ---- ZApp/App/_States/ZAppSequenceRunning.TcPOU
FUNCTION_BLOCK ZAppSequenceRunning EXTENDS ZAppSequence IMPLEMENTS ZCore.ISequence
VAR
  _step : ZCore.Step(ZAppStep.RunningBegin, ZAppStep.RunningEnd);
END_VAR

IF OnStart(_step)
THEN
  // init custom sequence variables here ...
END_IF

REPEAT
  LogStep();

  CASE _step.Index OF
    (* -------------------------------------------------------------------------------------------------------------------------------- *)
    ZAppStep.RunningBegin:
    (* -------------------------------------------------------------------------------------------------------------------------------- *)
      ; // implement me
      
    (* -------------------------------------------------------------------------------------------------------------------------------- *)
    ZAppStep.RunningEnd:
    (* -------------------------------------------------------------------------------------------------------------------------------- *)
      SetBusy(FALSE);
      
  ELSE
    Abort('sequence contains unhandled step');
  END_CASE
UNTIL _step.IsNotRepeatable() OR_ELSE NOT Busy END_REPEAT

END_FUNCTION_BLOCK

// ---- ZApp/Unit/Transport/TransportUnit.TcPOU
/// Declaration of a distinct unit of this application
FUNCTION_BLOCK TransportUnit EXTENDS ZApplication.Unit IMPLEMENTS ITransport, ZAux.IStateMachineListener
VAR
  _equipment : TransportEquipment(THIS^);
  _data : TransportDataRef;
  _com : TransportComRef;

  _boot : TransportSequenceBoot(THIS^);
  _automatic : TransportSequenceAutomatic(THIS^);
  _stop : TransportSequenceStop(THIS^);
  _gohome : TransportSequenceGoHome(THIS^);
  _faultReaction : TransportSequenceFaultReaction(THIS^);
  
  _statemachine : ZApplication.UnitStateMachine;

  _observeTimer : ZAux.Timer;
END_VAR

{attribute 'ZId' := '086a579c-dc1b-407f-8e70-5b7d4742c739'}

IF _observeTimer.Done THEN
  _observeTimer.WaitAsync(0.1);
  
  // monitor _com for requested actions (e.g. start homing, start automatic mode, ...)
  ObserveRequest(_com.Subscribe.Request.Start, ZApplication.UnitStateMachineState.Automatic);
  ObserveRequest(_com.Subscribe.Request.Stop, ZApplication.UnitStateMachineState.Stop);
  ObserveRequest(_com.Subscribe.Request.GoHome, ZApplication.UnitStateMachineState.GoHome);
  ObserveRequest(_com.Subscribe.Request.Halt, ZApplication.UnitStateMachineState.Halt);
  
  // provide relevant information via ADS
  _com.Publish.Request.Stop := _stateMachine.IsTransitionAllowed(ZApplication.UnitStateMachineState.Stop);
  _com.Publish.Request.Start := _stateMachine.IsTransitionAllowed(ZApplication.UnitStateMachineState.Automatic);
  _com.Publish.Request.GoHome := _stateMachine.IsTransitionAllowed(ZApplication.UnitStateMachineState.GoHome);
  _com.Publish.Request.Halt := _stateMachine.IsTransitionAllowed(ZApplication.UnitStateMachineState.Halt);

  _com.Publish.State := _stateMachine.State();
END_IF

METHOD FB_init : BOOL
VAR_INPUT
  bInitRetains : BOOL; // if TRUE, the retain variables are initialized (warm start / cold start)
  bInCopyCode : BOOL;  // if TRUE, the instance afterwards gets moved into the copy code (online change)
  parent : ZCore.IManagedObject; // caller of the Unit's cyclic method. If the Unit runs in its own context use 0
  name : ZCore.ZString;  // name of this unit as it should show up in the logger
  configdata : REFERENCE TO TransportDataConfig;  // reference to the configuration data that is used during boot to configure the Units equipment
  machinedata : REFERENCE TO TransportDataMachine; // reference to the machine data that is used through most sequences of the unit (motor speed, axes positions, ...)
  calibrationdata : REFERENCE TO TransportDataCalibration;  // reference to calibration that is determined by calibration sequences of the unit (static offsets, shifts)
  com : REFERENCE TO TransportCom;  // reference to the communication interface that is used to control this Unit via ADS
END_VAR
_name := name;

// initialize local logger decorator
_loggerDecorator.FB_init(bInitRetains, bInCopyCode, name, ZModuleProgram.Logger);
_alarmingDecorator.FB_init(bInitRetains, bInCopyCode, name, ZModuleProgram.Alarming);

// setup data
_data.Config REF= configdata;
_data.Machine REF= machinedata;
_data.Calibration REF= calibrationdata;
_com.Publish REF= com.Publish;
_com.Subscribe REF= com.Subscribe;

// ------- sequence initialization, map sequences of this unit to the statemachine -------
{attribute '__ZwPlcUnitInitSequenceImplementation__'} // Do not remove this attribute! It is used for code generation.
_statemachine.SetSequence(ZApplication.UnitStateMachineState.Boot, _boot);
_statemachine.SetSequence(ZApplication.UnitStateMachineState.FaultReaction, _faultReaction);
_statemachine.SetSequence(ZApplication.UnitStateMachineState.Gohome, _gohome);
_statemachine.SetSequence(ZApplication.UnitStateMachineState.Stop, _stop);
_statemachine.SetSequence(ZApplication.UnitStateMachineState.Automatic, _automatic);

_statemachine.SetName(_name);
_statemachine.SetListener(THIS^);
_statemachine.SetLogger(_logger);

// set initial state
_statemachine.SetState(ZApplication.UnitStateMachineState.Boot);
_statemachineIntrf := _statemachine;
END_METHOD

/// This method is called by a [Statemachine's startTransition method](xref:ZApplication.UnitStateMachine#startTransition)
/// if a given transition was failed (e.g. the transition is not allowed according to the state diagram of the state machine).
/// The State that was active previously in the StateMachine remains active and `requestedState` indicates which state transition
/// was requested by the user.
METHOD OnStartTransitionFailed
VAR_INPUT
  state : INT;  
  requestedState : INT;
END_VAR
END_METHOD

/// This method is called by a [Statemachine's startTransition method](xref:ZApplication.UnitStateMachine#startTransition)
/// if a given transition was successful. Please note, that at the time this event occurs, `state` still holds the
/// state that was active before calling `startTransition`, there is still one more call to this `state` to allow it to 
/// cleanup.
METHOD OnStartTransitionSucceeded
VAR_INPUT
  state : INT;  
  newState : INT;
END_VAR
END_METHOD

/// This method is called after a transition succeeded, right before the [start method of a sequence](xref:ZAux#start) is called.
/// The parameter `state` indicates the State that is active in the statemachine.
METHOD OnStateEntry
VAR_INPUT
  state : INT;
END_VAR
END_METHOD

/// This method is called after a sequence reported an error, but before the state machine starts its error handling.
METHOD OnStateError
VAR_INPUT
  state : INT;
END_VAR
END_METHOD

/// This method is called after a transition succeeded, right before the [stop method of a sequence](xref:ZAux#start) is called.
/// The parameter `state` indicates the State that is active in the statemachine.
METHOD OnStateExit
VAR_INPUT
  state : INT;  
END_VAR
END_METHOD

/// This method if a State has been executed successfully.
/// The parameter `state` indicates the State that is active in the statemachine.
METHOD OnStateSuccess
VAR_INPUT
  state : INT;    
END_VAR
END_METHOD

END_FUNCTION_BLOCK

// ---- ZApp/Unit/Transport/_Equipment/TransportEquipment.TcPOU
/// This function block is a container for equipment that is used by this unit.
/// Equipment is grouped by its kind (actuator, axes, io, ...).
/// It extends from [ManagedObjectContainer](xref:ZCore.ManagedObjectContainer) such that the parent
/// (= the unit itself) can be passed to equipment instances.
FUNCTION_BLOCK TransportEquipment EXTENDS TransportContainer
VAR_INPUT
  Io : TransportIo(_parent);
  Actuator : TransportActuator(_parent);
  Axis : TransportAxis(_parent);
  Fieldbus : TransportFieldbus(_parent);
  Unit : TransportLinkedUnit(_parent);
END_VAR

END_FUNCTION_BLOCK

// ---- ZApp/Unit/Transport/_SubObjects/TransportContainer.TcPOU
FUNCTION_BLOCK TransportContainer EXTENDS ZCore.ObjectContainer
VAR_INPUT
END_VAR
VAR_OUTPUT
END_VAR
VAR
  {attribute 'hide'}
  _parent : REFERENCE TO TransportUnit;
END_VAR

{ attribute 'hide' }
METHOD FB_init : BOOL
VAR_INPUT
	bInitRetains : BOOL; // if TRUE, the retain variables are initialized (warm start / cold start)
	bInCopyCode : BOOL;  // if TRUE, the instance afterwards gets moved into the copy code (online change)
  unit : REFERENCE TO TransportUnit;
END_VAR
_parent REF= unit;
END_METHOD

END_FUNCTION_BLOCK

// ---- ZApp/Unit/Transport/_Equipment/TransportIo.TcPOU
/// This function block is a container for all I/Os that are used by this unit.
/// The parent of all objects can be directly transfered in their constructor (this is only relevant for equipment objects
/// that have to be managed (e.g. [DebouncedInput](xref:ZEquipment.DebouncedInput), [Light](xref:ZEquipment.Light), ...).
FUNCTION_BLOCK TransportIo EXTENDS TransportContainer
VAR
  {attribute 'hide'}
  _iobridge : ZApplication.IoBridge(_parent);
END_VAR
VAR_INPUT

{attribute '__ZwPlcUnitEquipmentDeclaration__'} // Do not remove this attribute! It is used for code generation.
END_VAR

IF _isInitialized
THEN
  RETURN;
END_IF

  _iobridge.SetLogger(_parent._logger);

{attribute '__ZwPlcUnitEquipmentImplementation__'} // Do not remove this attribute! It is used for code generation.

_isInitialized := TRUE;

END_FUNCTION_BLOCK

// ---- ZApp/Unit/Transport/_Equipment/TransportActuator.TcPOU
/// This function block is a container for all actuator objects that are used by this unit.
/// The parent of all objects can be directly transfered in their constructor (this is only relevant for equipment objects
/// that have to be managed (e.g. [DebouncedInput](xref:ZEquipment.DebouncedInput), [Light](xref:ZEquipment.Light), ...).
FUNCTION_BLOCK TransportActuator EXTENDS TransportContainer
VAR
  {attribute 'hide'}
  _actuatorbridge : ZApplication.ActuatorBridge(_parent);
  {attribute 'hide'}
  _iobridge : ZApplication.IoBridge(_parent);
END_VAR
VAR_INPUT

{region "Gripper : ActuatorDigitalBiLsPlusMinus"}
  Gripper : TransportActuatorGripper(_parent);
  {attribute 'ZId' := '5d1fe583-4573-4e37-9380-49c474c02543'}
{endregion}

{attribute '__ZwPlcUnitEquipmentDeclaration__'} // Do not remove this attribute! It is used for code generation.
END_VAR

IF _isInitialized
THEN
  RETURN;
END_IF

  _actuatorbridge.SetLogger(_parent._logger);

{region "Gripper : ActuatorDigitalBiLsPlusMinus"}
  Gripper.SetLogger(_parent._logger);
  Gripper.SetName(name:='Gripper', movePlusName:='Open', moveMinusName:='Close', plusName:='IsOpen', minusName:='IsClosed');
  Gripper.SetSimulation(SEL(_parent._data.Config.Simulated, ActuatorDigitalSimulation.Disabled, ZEquipment.ActuatorDigitalSimulation.Automatic));
  Gripper.SetSimulationUncertainty(uncertainty:=10);
  Gripper.SetDelay(plusStartDuration:=0, plusEndDuration:=0, minusStartDuration:=0, minusEndDuration:=0, stop:=0);
  Gripper.SetSwitchDuration(plusDuration:=0.2, minusDuration:=0.2);
  Gripper.SetMovementDuration(plusDuration:=3, minusDuration:=3);
  Gripper.SetTimeout(plusDuration:=5, minusDuration:=5);
  _actuatorbridge.AddActuatorDigital(Gripper, publish := _parent._com.Publish.Equipment.Gripper, subscribe := _parent._com.Subscribe.Equipment.Gripper);
  _iobridge.AddDigitalOutput(Gripper.MinusOutput, publish := _parent._com.Publish.Equipment.GripperClose, subscribe := _parent._com.Subscribe.Equipment.GripperClose);
  _iobridge.AddDigitalOutput(Gripper.PlusOutput, publish := _parent._com.Publish.Equipment.GripperOpen, subscribe := _parent._com.Subscribe.Equipment.GripperOpen);
  _iobridge.AddDigitalInput(Gripper.MinusInput, publish := _parent._com.Publish.Equipment.GripperIsClosed, subscribe := _parent._com.Subscribe.Equipment.GripperIsClosed);
  _iobridge.AddDigitalInput(Gripper.PlusInput, publish := _parent._com.Publish.Equipment.GripperIsOpen, subscribe := _parent._com.Subscribe.Equipment.GripperIsOpen);
  {region "UserInitCode"}
  // put your individual init code for this Actuator here
  {endregion}

  {attribute 'ZId' := '5d1fe583-4573-4e37-9380-49c474c02543'}
{endregion}

{attribute '__ZwPlcUnitEquipmentImplementation__'} // Do not remove this attribute! It is used for code generation.

_isInitialized := TRUE;

END_FUNCTION_BLOCK

// ---- ZApp/Unit/Transport/_Equipment/TransportActuatorGripper.TcPOU
FUNCTION_BLOCK TransportActuatorGripper EXTENDS ZEquipment.ActuatorDigitalBiLsPlusMinus

METHOD PUBLIC CloseAsync
VAR_INPUT
  startToken : ZCore.IStartToken;
END_VAR
MoveMinusAsync(startToken:=startToken);
END_METHOD

METHOD PUBLIC IsClosed : BOOL
VAR_INPUT
END_VAR
IsClosed := IsAtMinus();
END_METHOD

METHOD PUBLIC IsOpen : BOOL
VAR_INPUT
END_VAR
IsOpen := IsAtPlus();
END_METHOD

METHOD PUBLIC OpenAsync
VAR_INPUT
  startToken : ZCore.IStartToken;
END_VAR
MovePlusAsync(startToken:=startToken);
END_METHOD

END_FUNCTION_BLOCK

// ---- ZApp/Unit/Transport/_Equipment/TransportAxis.TcPOU
/// This function block is a container for all axis objects that are used by this unit.
/// The parent of all objects can be directly transfered in their constructor (this is only relevant for equipment objects
/// that have to be managed (e.g. [DebouncedInput](xref:ZEquipment.DebouncedInput), [Light](xref:ZEquipment.Light), ...).
FUNCTION_BLOCK TransportAxis EXTENDS TransportContainer
VAR
  {attribute 'hide'}
  _axisbridge : ZApplication.AxisBridge(_parent);
END_VAR
VAR_INPUT

{region "HorizontalX : AxisPlcOpenMc"}
  HorizontalX : ZEquipment.AxisPlcOpenMc(_parent);
  {attribute 'ZId' := 'b48886d3-effd-43af-8c1e-4c35e310bf5b'}
{endregion}

{region "VerticalZ : AxisPlcOpenMc"}
  VerticalZ : ZEquipment.AxisPlcOpenMc(_parent);
  {attribute 'ZId' := '82c3e667-8dc4-4ea4-a1fc-9c83583bfea0'}
{endregion}

{attribute '__ZwPlcUnitEquipmentDeclaration__'} // Do not remove this attribute! It is used for code generation.
END_VAR

IF _isInitialized
THEN
  RETURN;
END_IF

  _axisbridge.SetLogger(_parent._logger);

{region "HorizontalX : AxisPlcOpenMc"}
  HorizontalX.SetLogger(_parent._logger);
  HorizontalX.SetName(name:='HorizontalX');
  HorizontalX.SetSimulation(_parent._data.Config.Simulated);
  _axisbridge.AddAxisPlcOpenMc(axis:=HorizontalX, publish:=_parent._com.Publish.Equipment.HorizontalX, subscribe:=_parent._com.Subscribe.Equipment.HorizontalX);

  {region "UserInitCode"}
  // put your individual init code for this Axis here
  {endregion}

  {attribute 'ZId' := 'b48886d3-effd-43af-8c1e-4c35e310bf5b'}
{endregion}

{region "VerticalZ : AxisPlcOpenMc"}
  VerticalZ.SetLogger(_parent._logger);
  VerticalZ.SetName(name:='VerticalZ');
  VerticalZ.SetSimulation(_parent._data.Config.Simulated);
  _axisbridge.AddAxisPlcOpenMc(axis:=VerticalZ, publish:=_parent._com.Publish.Equipment.VerticalZ, subscribe:=_parent._com.Subscribe.Equipment.VerticalZ);

  {region "UserInitCode"}
  // put your individual init code for this Axis here
  {endregion}

  {attribute 'ZId' := '82c3e667-8dc4-4ea4-a1fc-9c83583bfea0'}
{endregion}

{attribute '__ZwPlcUnitEquipmentImplementation__'} // Do not remove this attribute! It is used for code generation.

_isInitialized := TRUE;

END_FUNCTION_BLOCK

// ---- ZApp/Unit/Transport/_Equipment/TransportFieldbus.TcPOU
/// This function block is a container for all axis objects that are used by this unit.
/// The parent of all objects can be directly transfered in their constructor (this is only relevant for equipment objects
/// that have to be managed (e.g. [DebouncedInput](xref:ZEquipment.DebouncedInput), [Light](xref:ZEquipment.Light), ...).
FUNCTION_BLOCK TransportFieldbus EXTENDS TransportContainer
VAR
END_VAR
VAR_INPUT

{attribute '__ZwPlcUnitEquipmentDeclaration__'} // Do not remove this attribute! It is used for code generation.
END_VAR

IF _isInitialized
THEN
  RETURN;
END_IF

{attribute '__ZwPlcUnitEquipmentImplementation__'} // Do not remove this attribute! It is used for code generation.

_isInitialized := TRUE;

END_FUNCTION_BLOCK

// ---- ZApp/Unit/Transport/_Equipment/TransportLinkedUnit.TcPOU
/// This function block is a container for all linked units that are used by this unit.
/// Linked units can be addressed through their individual interface.
FUNCTION_BLOCK TransportLinkedUnit EXTENDS TransportContainer
VAR_INPUT
  Assembly : IAssembly;
  Drilling : IDrilling;
  QualityInspection : IQualityInspection;
{attribute '__ZwPlcUnitEquipmentDeclaration__'} // Do not remove this attribute! It is used for code generation.
END_VAR

IF _isInitialized
THEN
  RETURN;
END_IF

Assembly := ZModuleProgram.Assembly;
Drilling := ZModuleProgram.Drilling;
QualityInspection := ZModuleProgram.QualityInspection;

{attribute '__ZwPlcUnitEquipmentImplementation__'} // Do not remove this attribute! It is used for code generation.

_isInitialized := TRUE;

END_FUNCTION_BLOCK

// ---- ZApp/Unit/Transport/_States/TransportSequenceBoot.TcPOU
FUNCTION_BLOCK TransportSequenceBoot EXTENDS TransportSequence IMPLEMENTS ZCore.ISequence
VAR
  _step : ZCore.Step(TransportStep.BootBegin, TransportStep.BootEnd);
END_VAR

IF OnStart(_step) THEN
  ; // init custom sequence variables here ...
END_IF

REPEAT
  LogStep();

  CASE _step.Index OF
    (* -------------------------------------------------------------------------------------------------------------------------------- *)
    TransportStep.BootBegin:
    (* -------------------------------------------------------------------------------------------------------------------------------- *)
      IF _step.OnEntry()
      THEN
        // initialize equipment
        _io();
        _actuator();
        _fieldbus();
        _axis();
        _unit();
      END_IF
      
      _parent._objectManager.Cyclic();      
      Assert(_parent._objectManager);
      IF _parent._objectManager.Done
      THEN
        _step.SetNext(TransportStep.BootEnd);
      END_IF

    (* -------------------------------------------------------------------------------------------------------------------------------- *)
    TransportStep.BootEnd:
    (* -------------------------------------------------------------------------------------------------------------------------------- *)
      SetBusy(FALSE);
      
  ELSE
    Abort('sequence contains unhandled step');
  END_CASE
UNTIL _step.IsNotRepeatable() OR_ELSE NOT Busy END_REPEAT

END_FUNCTION_BLOCK

// ---- ZApp/Unit/Transport/_SubObjects/TransportSequence.TcPOU
FUNCTION_BLOCK TransportSequence EXTENDS ZApplication.Sequence
VAR
  {attribute 'hide'}
  _parent : REFERENCE TO TransportUnit;
  _io : REFERENCE TO TransportIo;
  _actuator : REFERENCE TO TransportActuator;
  _fieldbus : REFERENCE TO TransportFieldbus;
  _axis : REFERENCE TO TransportAxis;
  _data : REFERENCE TO TransportDataRef;
  _unit : REFERENCE TO TransportLinkedUnit;  
END_VAR

METHOD FB_init : BOOL
VAR_INPUT
  bInitRetains : BOOL; // if TRUE, the retain variables are initialized (warm start / cold start)
  bInCopyCode : BOOL;  // if TRUE, the instance afterwards gets moved into the copy code (online change)
  unit : REFERENCE TO TransportUnit;
END_VAR
_parent REF= unit;
_alarming := unit._alarming;
_io REF= unit._equipment.Io;
_actuator REF= unit._equipment.Actuator;
_fieldbus REF= unit._equipment.Fieldbus;
_axis REF= unit._equipment.Axis;
_unit REF= unit._equipment.Unit;
_data REF= unit._data;
_loggerDiagnostics.SetLogger(unit._logger);
END_METHOD

METHOD StepDecoded : ZCore.ZString
VAR_INPUT
  stepIndex : INT;
END_VAR
VAR_INST
  _stepIndexDecoded : TransportStep;
END_VAR
_stepIndexDecoded := stepIndex;
stepDecoded := TO_STRING(_stepIndexDecoded);
END_METHOD

END_FUNCTION_BLOCK

// ---- ZApp/Unit/Transport/_States/TransportSequenceAutomatic.TcPOU
FUNCTION_BLOCK TransportSequenceAutomatic EXTENDS TransportSequence IMPLEMENTS ZCore.ISequence
VAR
  _step : ZCore.Step(TransportStep.AutomaticBegin, TransportStep.AutomaticEnd);
  _timer : ZAux.Timer;
END_VAR

IF NOT Busy THEN
  RETURN;
END_IF

IF OnStart(_step) THEN
  ; // init custom sequence variables here ...
END_IF

IF OnStop() THEN
  RETURN; // external stop was triggered
END_IF

IF OnHalt() THEN
  Halting := TRUE;
END_IF

REPEAT
  LogStep();

  CASE _step.Index OF
    (* -------------------------------------------------------------------------------------------------------------------------------- *)
    TransportStep.AutomaticBegin:
    (* -------------------------------------------------------------------------------------------------------------------------------- *)
      IF _step.OnEntry()
      THEN
        ;
      END_IF

      _step.SetNext(TransportStep.AutomaticInitializeMovements);

    (* -------------------------------------------------------------------------------------------------------------------------------- *)
    TransportStep.AutomaticInitializeMovements:
    (* -------------------------------------------------------------------------------------------------------------------------------- *)
      IF _step.OnEntry()
      THEN        
        _timer.WaitAsync(1.2);
        _logger.Info('Init Movements!');
      END_IF
      
      Await(obj1:=_timer, nextStep:=TransportStep.AutomaticMoveToLeftPos);

    (* -------------------------------------------------------------------------------------------------------------------------------- *)
    TransportStep.AutomaticMoveToLeftPos:
    (* -------------------------------------------------------------------------------------------------------------------------------- *)
      IF _step.OnEntry()
      THEN        
        _axis.HorizontalX.MoveAbsoluteAsync(startToken:=THIS^, position:=_data.Machine.HorizontalLeftPos, speed:=_data.Machine.Highspeed);
      END_IF
      
      Await(obj1:=_axis.HorizontalX, nextStep:=TransportStep.AutomaticWaitSomeTime);

    (* -------------------------------------------------------------------------------------------------------------------------------- *)
    TransportStep.AutomaticWaitSomeTime:
    (* -------------------------------------------------------------------------------------------------------------------------------- *)
      IF _step.OnEntry()
      THEN
        Milestone('Standing on the left side, halt may occur');
        
        IF Halting 
        THEN
          _step.SetNext(TransportStep.AutomaticEnd);
          RETURN;        
        ELSE
          _timer.WaitAsync(2.0);
        END_IF  
      END_IF
      
      Await(obj1:=_timer, nextStep:=TransportStep.AutomaticMoveVerticalDown);

    (* -------------------------------------------------------------------------------------------------------------------------------- *)
    TransportStep.AutomaticMoveVerticalDown:
    (* -------------------------------------------------------------------------------------------------------------------------------- *)
      IF _step.OnEntry()
      THEN        
        _axis.VerticalZ.MoveAbsoluteAsync(startToken:=THIS^, position:=_data.Machine.VerticalBottomPos, speed:=_data.Machine.Highspeed);
      END_IF
      
      Await(obj1:=_axis.VerticalZ, nextStep:=TransportStep.AutomaticCloseGripper);

    (* -------------------------------------------------------------------------------------------------------------------------------- *)
    TransportStep.AutomaticCloseGripper:
    (* -------------------------------------------------------------------------------------------------------------------------------- *)
      IF _step.OnEntry()
      THEN        
        _actuator.Gripper.CloseAsync(startToken:=THIS^);
      END_IF
      
      Await(obj1:=_actuator.Gripper, nextStep:=TransportStep.AutomaticMoveVerticalToTopPos);

    (* -------------------------------------------------------------------------------------------------------------------------------- *)
    TransportStep.AutomaticMoveVerticalToTopPos:
    (* -------------------------------------------------------------------------------------------------------------------------------- *)
      IF _step.OnEntry()
      THEN        
        _axis.VerticalZ.MoveAbsoluteAsync(startToken:=THIS^, position:=_data.Machine.VerticalTopPos, speed:=_data.Machine.Highspeed);
      END_IF
      
      Await(obj1:=_axis.VerticalZ, nextStep:=TransportStep.AutomaticWaitSomeMoreTime);

    (* -------------------------------------------------------------------------------------------------------------------------------- *)
    TransportStep.AutomaticWaitSomeMoreTime:
    (* -------------------------------------------------------------------------------------------------------------------------------- *)
      IF _step.OnEntry()
      THEN        
        Milestone('Standing on the top with closed gripper, halt may occur!');
        
        IF Halting 
        THEN
          _step.SetNext(TransportStep.AutomaticEnd);
          RETURN;        
        ELSE
          _timer.WaitAsync(2.0);
        END_IF  
      END_IF
      
      Await(obj1:=_timer, nextStep:=TransportStep.AutomaticMoveToCamPos);

    (* -------------------------------------------------------------------------------------------------------------------------------- *)
    TransportStep.AutomaticMoveToCamPos:
    (* -------------------------------------------------------------------------------------------------------------------------------- *)
      IF _step.OnEntry()
      THEN        
        _axis.HorizontalX.MoveAbsoluteAsync(startToken:=THIS^, position:=_data.Machine.HorizontalCamPos, speed:=_data.Machine.Highspeed);
      END_IF
      
      Await(obj1:=_axis.HorizontalX, nextStep:=TransportStep.AutomaticStartQualityInspection);    

    (* -------------------------------------------------------------------------------------------------------------------------------- *)
    TransportStep.AutomaticStartQualityInspection:
    (* -------------------------------------------------------------------------------------------------------------------------------- *)
      IF _step.OnEntry()
      THEN        
        _unit.QualityInspection.RunAutomaticAsync(startToken:=THIS^, unit:=_parent);
      END_IF
      
      IF _unit.QualityInspection.Error
      THEN
        Abort(_unit.QualityInspection.ErrorMessage());
      ELSIF NOT _unit.QualityInspection.Busy
      THEN
        _unit.QualityInspection.Unlock(unit:=_parent);
        _step.SetNext(TransportStep.AutomaticMoveToRightPos);
			END_IF
      
    (* -------------------------------------------------------------------------------------------------------------------------------- *)
    TransportStep.AutomaticMoveToRightPos:
    (* -------------------------------------------------------------------------------------------------------------------------------- *)
      IF _step.OnEntry()
      THEN        
        _axis.HorizontalX.MoveAbsoluteAsync(startToken:=THIS^, position:=_data.Machine.HorizontalRightPos, _data.Machine.Highspeed);
      END_IF
      
      Await(obj1:=_axis.HorizontalX, nextStep:=TransportStep.AutomaticOpenGripper);

    (* -------------------------------------------------------------------------------------------------------------------------------- *)
    TransportStep.AutomaticOpenGripper:
    (* -------------------------------------------------------------------------------------------------------------------------------- *)
      IF _step.OnEntry()
      THEN        
        _actuator.Gripper.OpenAsync(startToken:=THIS^);
      END_IF
      
      IF Halting
      THEN
        Await(obj1:=_actuator.Gripper, nextStep:=TransportStep.AutomaticCleanUp);
      ELSE
        Await(obj1:=_actuator.Gripper, nextStep:=TransportStep.AutomaticInitializeMovements);
      END_IF

    (* -------------------------------------------------------------------------------------------------------------------------------- *)
    TransportStep.AutomaticCleanUp:
    (* -------------------------------------------------------------------------------------------------------------------------------- *)
      IF _step.OnEntry()
      THEN        
        _timer.WaitAsync(1.0);
        _logger.Info('Waiting some time -> Halt occured');
      END_IF
      
      Await(obj1:=_timer, nextStep:=TransportStep.AutomaticEnd);
    
    (* -------------------------------------------------------------------------------------------------------------------------------- *)
    TransportStep.AutomaticEnd:
    (* -------------------------------------------------------------------------------------------------------------------------------- *)
      SetBusy(FALSE);
  
  ELSE
    Abort('sequence contains unhandled step');
  END_CASE
UNTIL _step.IsNotRepeatable() OR_ELSE NOT Busy END_REPEAT

END_FUNCTION_BLOCK

// ---- ZApp/Unit/Transport/_States/TransportSequenceStop.TcPOU
FUNCTION_BLOCK TransportSequenceStop EXTENDS TransportSequence IMPLEMENTS ZCore.ISequence
VAR
  _step : ZCore.Step(TransportStep.StopBegin, TransportStep.StopEnd);
  _timerSim : ZAux.Timer;
END_VAR

IF OnStart(_step) THEN
  ; // init custom sequence variables here ...
END_IF

REPEAT
  LogStep();

  CASE _step.Index OF
    (* -------------------------------------------------------------------------------------------------------------------------------- *)
    TransportStep.StopBegin:
    (* -------------------------------------------------------------------------------------------------------------------------------- *)
      IF _step.OnEntry()
      THEN
        _axis.HorizontalX.StopAsync(startToken:=THIS^);
        _axis.VerticalZ.StopAsync(startToken:=THIS^);
			END_IF
      
      Await2(obj1:=_axis.HorizontalX, obj2:=_axis.VerticalZ, nextStep:=TransportStep.StopEnd);

    (* -------------------------------------------------------------------------------------------------------------------------------- *)
    TransportStep.StopEnd:
    (* -------------------------------------------------------------------------------------------------------------------------------- *)    
      SetBusy(FALSE);
  
  ELSE
    Abort('sequence contains unhandled step');
  END_CASE
UNTIL _step.IsNotRepeatable() OR_ELSE NOT Busy END_REPEAT

END_FUNCTION_BLOCK

// ---- ZApp/Unit/Transport/_States/TransportSequenceGoHome.TcPOU
FUNCTION_BLOCK TransportSequenceGoHome EXTENDS TransportSequence IMPLEMENTS ZCore.ISequence
VAR
  _step : ZCore.Step(TransportStep.GohomeBegin, TransportStep.GohomeEnd);
  _timer : ZAux.Timer;
END_VAR

IF NOT Busy THEN
  RETURN;
END_IF

IF OnStart(_step) THEN
  ; // init custom sequence variables here ...
END_IF

IF OnStop() THEN
  RETURN; // external stop was triggered
END_IF

IF OnHalt() THEN
  ; // Halting := TRUE; // Uncomment to acknowledge that the sequence is halting
END_IF

REPEAT
  LogStep();

  CASE _step.Index OF
    (* -------------------------------------------------------------------------------------------------------------------------------- *)
    TransportStep.GoHomeBegin:
    (* -------------------------------------------------------------------------------------------------------------------------------- *)
      IF _step.OnEntry()
      THEN
        _timer.WaitAsync(2);
			END_IF
      
      Await(_timer, nextStep:=TransportStep.GoHomeVerticalUp);

    (* -------------------------------------------------------------------------------------------------------------------------------- *)
    TransportStep.GoHomeVerticalUp:
    (* -------------------------------------------------------------------------------------------------------------------------------- *)
      IF _step.OnEntry()
      THEN        
        _axis.VerticalZ.MoveAbsoluteAsync(startToken:=THIS^, position:=_data.Machine.VerticalHomePos, speed:=_data.Machine.Slowspeed);
      END_IF
      
      Await(obj1:=_axis.VerticalZ, nextStep:=TransportStep.GoHomeHorizontalToRightPos);

    (* -------------------------------------------------------------------------------------------------------------------------------- *)
    TransportStep.GoHomeHorizontalToRightPos:
    (* -------------------------------------------------------------------------------------------------------------------------------- *)
      IF _step.OnEntry()
      THEN        
        _axis.HorizontalX.MoveAbsoluteAsync(startToken:=THIS^, position:=_data.Machine.HorizontalHomePos, speed:=_data.Machine.Slowspeed);
      END_IF
      
      Await(obj1:=_axis.HorizontalX, nextStep:=TransportStep.GoHomeUnlockQualityInspection);

    (* -------------------------------------------------------------------------------------------------------------------------------- *)
    TransportStep.GoHomeUnlockQualityInspection:
    (* -------------------------------------------------------------------------------------------------------------------------------- *)
      _unit.QualityInspection.Unlock(unit:=_parent);
      _step.SetNext(index:=TransportStep.GoHomeStartHomingOfChilds);

    (* -------------------------------------------------------------------------------------------------------------------------------- *)
    TransportStep.GoHomeStartHomingOfChilds:
    (* -------------------------------------------------------------------------------------------------------------------------------- *)
      IF _step.OnEntry()
      THEN        
        _unit.Assembly.HomingAsync(startToken:=THIS^, unit:=0); // <- For homing we do not need to lock, therefore 0 on second parameter)
        _unit.Drilling.HomingAsync(startToken:=THIS^, unit:=0);
        _unit.QualityInspection.HomingAsync(THIS^, 0);
      END_IF
      
      Await3(obj1:=_unit.Assembly, obj2:=_unit.Drilling, obj3:=_unit.QualityInspection, nextStep:=TransportStep.GoHomeEnd);

    (* -------------------------------------------------------------------------------------------------------------------------------- *)
    TransportStep.GoHomeEnd:
    (* -------------------------------------------------------------------------------------------------------------------------------- *)
      SetBusy(FALSE);
  
  ELSE
    Abort('sequence contains unhandled step');
  END_CASE
UNTIL _step.IsNotRepeatable() OR_ELSE NOT Busy END_REPEAT

END_FUNCTION_BLOCK

// ---- ZApp/Unit/Transport/_States/TransportSequenceFaultReaction.TcPOU
FUNCTION_BLOCK TransportSequenceFaultReaction EXTENDS TransportSequence IMPLEMENTS ZCore.ISequence
VAR
  _step : ZCore.Step(TransportStep.FaultReactionBegin, TransportStep.FaultReactionEnd);
  _timerSim : ZAux.Timer;
END_VAR

IF OnStart(_step) THEN
  ; // init custom sequence variables here ...
END_IF

REPEAT
  LogStep();

  CASE _step.Index OF
    (* -------------------------------------------------------------------------------------------------------------------------------- *)
    TransportStep.FaultReactionBegin:
    (* -------------------------------------------------------------------------------------------------------------------------------- *)
      IF _step.OnEntry()
      THEN
        _axis.HorizontalX.StopAsync(startToken:=THIS^);
        _axis.VerticalZ.StopAsync(startToken:=THIS^);
			END_IF
      
      Await2(obj1:=_axis.HorizontalX, obj2:=_axis.VerticalZ, nextStep:=TransportStep.FaultReactionVerticalUp);

    (* -------------------------------------------------------------------------------------------------------------------------------- *)
    TransportStep.FaultReactionVerticalUp:
    (* -------------------------------------------------------------------------------------------------------------------------------- *)
      IF _step.OnEntry()
      THEN        
        _axis.VerticalZ.MoveAbsoluteAsync(startToken:=THIS^, position:=_data.Machine.VerticalTopPos, speed:=_data.Machine.Slowspeed);
      END_IF
      
      Await(obj1:=_axis.VerticalZ, nextStep:=TransportStep.FaultReactionEnd);

    (* -------------------------------------------------------------------------------------------------------------------------------- *)
    TransportStep.FaultReactionEnd:
    (* -------------------------------------------------------------------------------------------------------------------------------- *)    
      SetBusy(FALSE);
  
  ELSE
    Abort('sequence contains unhandled step');
  END_CASE
UNTIL _step.IsNotRepeatable() OR_ELSE NOT Busy END_REPEAT

END_FUNCTION_BLOCK

// ---- ZApp/Unit/Drilling/DrillingUnit.TcPOU
/// Declaration of a distinct unit of this application
FUNCTION_BLOCK DrillingUnit EXTENDS ZApplication.Unit IMPLEMENTS IDrilling, ZAux.IStateMachineListener
VAR
  _equipment : DrillingEquipment(THIS^);
  _data : DrillingDataRef;
  _com : DrillingComRef;

  _boot : DrillingSequenceBoot(THIS^);
  _automatic : DrillingSequenceAutomatic(THIS^);
  _stop : DrillingSequenceStop(THIS^);
  _gohome : DrillingSequenceGoHome(THIS^);
  _faultReaction : DrillingSequenceFaultReaction(THIS^);
  
  _statemachine : ZApplication.UnitStateMachine;

  _observeTimer : ZAux.Timer;
END_VAR

{attribute 'ZId' := 'fb505b0c-135e-45db-86de-861c7673a58e'}

IF _observeTimer.Done THEN
  _observeTimer.WaitAsync(0.1);
  
  // monitor _com for requested actions (e.g. start homing, start automatic mode, ...)
  ObserveRequest(_com.Subscribe.Request.Start, ZApplication.UnitStateMachineState.Automatic);
  ObserveRequest(_com.Subscribe.Request.Stop, ZApplication.UnitStateMachineState.Stop);
  ObserveRequest(_com.Subscribe.Request.GoHome, ZApplication.UnitStateMachineState.GoHome);
  ObserveRequest(_com.Subscribe.Request.Halt, ZApplication.UnitStateMachineState.Halt);
  
  // provide relevant information via ADS
  _com.Publish.Request.Stop := _stateMachine.IsTransitionAllowed(ZApplication.UnitStateMachineState.Stop);
  _com.Publish.Request.Start := _stateMachine.IsTransitionAllowed(ZApplication.UnitStateMachineState.Automatic);
  _com.Publish.Request.GoHome := _stateMachine.IsTransitionAllowed(ZApplication.UnitStateMachineState.GoHome);
  _com.Publish.Request.Halt := _stateMachine.IsTransitionAllowed(ZApplication.UnitStateMachineState.Halt);

  _com.Publish.State := _stateMachine.State();
END_IF

METHOD FB_init : BOOL
VAR_INPUT
  bInitRetains : BOOL; // if TRUE, the retain variables are initialized (warm start / cold start)
  bInCopyCode : BOOL;  // if TRUE, the instance afterwards gets moved into the copy code (online change)
  parent : ZCore.IManagedObject; // caller of the Unit's cyclic method. If the Unit runs in its own context use 0
  name : ZCore.ZString;  // name of this unit as it should show up in the logger
  configdata : REFERENCE TO DrillingDataConfig;  // reference to the configuration data that is used during boot to configure the Units equipment
  machinedata : REFERENCE TO DrillingDataMachine; // reference to the machine data that is used through most sequences of the unit (motor speed, axes positions, ...)
  calibrationdata : REFERENCE TO DrillingDataCalibration;  // reference to calibration that is determined by calibration sequences of the unit (static offsets, shifts)
  com : REFERENCE TO DrillingCom;  // reference to the communication interface that is used to control this Unit via ADS
END_VAR
_name := name;

// initialize local logger decorator
_loggerDecorator.FB_init(bInitRetains, bInCopyCode, name, ZModuleProgram.Logger);
_alarmingDecorator.FB_init(bInitRetains, bInCopyCode, name, ZModuleProgram.Alarming);

// setup data
_data.Config REF= configdata;
_data.Machine REF= machinedata;
_data.Calibration REF= calibrationdata;
_com.Publish REF= com.Publish;
_com.Subscribe REF= com.Subscribe;

// ------- sequence initialization, map sequences of this unit to the statemachine -------
{attribute '__ZwPlcUnitInitSequenceImplementation__'} // Do not remove this attribute! It is used for code generation.
_statemachine.SetSequence(ZApplication.UnitStateMachineState.Boot, _boot);
_statemachine.SetSequence(ZApplication.UnitStateMachineState.FaultReaction, _faultReaction);
_statemachine.SetSequence(ZApplication.UnitStateMachineState.Gohome, _gohome);
_statemachine.SetSequence(ZApplication.UnitStateMachineState.Stop, _stop);
_statemachine.SetSequence(ZApplication.UnitStateMachineState.Automatic, _automatic);

_statemachine.SetName(_name);
_statemachine.SetListener(THIS^);
_statemachine.SetLogger(_logger);

// set initial state
_statemachine.SetState(ZApplication.UnitStateMachineState.Boot);
_statemachineIntrf := _statemachine;
END_METHOD

/// This method is called by a [Statemachine's startTransition method](xref:ZApplication.UnitStateMachine#startTransition)
/// if a given transition was failed (e.g. the transition is not allowed according to the state diagram of the state machine).
/// The State that was active previously in the StateMachine remains active and `requestedState` indicates which state transition
/// was requested by the user.
METHOD OnStartTransitionFailed
VAR_INPUT
  state : INT;  
  requestedState : INT;
END_VAR
END_METHOD

/// This method is called by a [Statemachine's startTransition method](xref:ZApplication.UnitStateMachine#startTransition)
/// if a given transition was successful. Please note, that at the time this event occurs, `state` still holds the
/// state that was active before calling `startTransition`, there is still one more call to this `state` to allow it to 
/// cleanup.
METHOD OnStartTransitionSucceeded
VAR_INPUT
  state : INT;  
  newState : INT;
END_VAR
END_METHOD

/// This method is called after a transition succeeded, right before the [start method of a sequence](xref:ZAux#start) is called.
/// The parameter `state` indicates the State that is active in the statemachine.
METHOD OnStateEntry
VAR_INPUT
  state : INT;
END_VAR
END_METHOD

/// This method is called after a sequence reported an error, but before the state machine starts its error handling.
METHOD OnStateError
VAR_INPUT
  state : INT;
END_VAR
END_METHOD

/// This method is called after a transition succeeded, right before the [stop method of a sequence](xref:ZAux#start) is called.
/// The parameter `state` indicates the State that is active in the statemachine.
METHOD OnStateExit
VAR_INPUT
  state : INT;  
END_VAR
END_METHOD

/// This method if a State has been executed successfully.
/// The parameter `state` indicates the State that is active in the statemachine.
METHOD OnStateSuccess
VAR_INPUT
  state : INT;    
END_VAR
END_METHOD

END_FUNCTION_BLOCK

// ---- ZApp/Unit/Drilling/_Equipment/DrillingEquipment.TcPOU
/// This function block is a container for equipment that is used by this unit.
/// Equipment is grouped by its kind (actuator, axes, io, ...).
/// It extends from [ManagedObjectContainer](xref:ZCore.ManagedObjectContainer) such that the parent
/// (= the unit itself) can be passed to equipment instances.
FUNCTION_BLOCK DrillingEquipment EXTENDS DrillingContainer
VAR_INPUT
  Io : DrillingIo(_parent);
  Actuator : DrillingActuator(_parent);
  Axis : DrillingAxis(_parent);
  Fieldbus : DrillingFieldbus(_parent);
  Unit : DrillingLinkedUnit(_parent);
END_VAR

END_FUNCTION_BLOCK

// ---- ZApp/Unit/Drilling/_SubObjects/DrillingContainer.TcPOU
FUNCTION_BLOCK DrillingContainer EXTENDS ZCore.ObjectContainer
VAR_INPUT
END_VAR
VAR_OUTPUT
END_VAR
VAR
  {attribute 'hide'}
  _parent : REFERENCE TO DrillingUnit;
END_VAR

{ attribute 'hide' }
METHOD FB_init : BOOL
VAR_INPUT
	bInitRetains : BOOL; // if TRUE, the retain variables are initialized (warm start / cold start)
	bInCopyCode : BOOL;  // if TRUE, the instance afterwards gets moved into the copy code (online change)
  unit : REFERENCE TO DrillingUnit;
END_VAR
_parent REF= unit;
END_METHOD

END_FUNCTION_BLOCK

// ---- ZApp/Unit/Drilling/_Equipment/DrillingIo.TcPOU
/// This function block is a container for all I/Os that are used by this unit.
/// The parent of all objects can be directly transfered in their constructor (this is only relevant for equipment objects
/// that have to be managed (e.g. [DebouncedInput](xref:ZEquipment.DebouncedInput), [Light](xref:ZEquipment.Light), ...).
FUNCTION_BLOCK DrillingIo EXTENDS DrillingContainer
VAR
  {attribute 'hide'}
  _iobridge : ZApplication.IoBridge(_parent);
END_VAR
VAR_INPUT

{attribute '__ZwPlcUnitEquipmentDeclaration__'} // Do not remove this attribute! It is used for code generation.
END_VAR

IF _isInitialized
THEN
  RETURN;
END_IF

  _iobridge.SetLogger(_parent._logger);

{attribute '__ZwPlcUnitEquipmentImplementation__'} // Do not remove this attribute! It is used for code generation.

_isInitialized := TRUE;

END_FUNCTION_BLOCK

// ---- ZApp/Unit/Drilling/_Equipment/DrillingActuator.TcPOU
/// This function block is a container for all actuator objects that are used by this unit.
/// The parent of all objects can be directly transfered in their constructor (this is only relevant for equipment objects
/// that have to be managed (e.g. [DebouncedInput](xref:ZEquipment.DebouncedInput), [Light](xref:ZEquipment.Light), ...).
FUNCTION_BLOCK DrillingActuator EXTENDS DrillingContainer
VAR
  {attribute 'hide'}
  _actuatorbridge : ZApplication.ActuatorBridge(_parent);
  {attribute 'hide'}
  _iobridge : ZApplication.IoBridge(_parent);
END_VAR
VAR_INPUT

{region "Vertical : ActuatorDigitalBiLsPlusMinus"}
  Vertical : DrillingActuatorVertical(_parent);
  {attribute 'ZId' := '6edc2aeb-8e0c-4ef7-9533-2d3679311649'}
{endregion}

{attribute '__ZwPlcUnitEquipmentDeclaration__'} // Do not remove this attribute! It is used for code generation.
END_VAR

IF _isInitialized
THEN
  RETURN;
END_IF

  _actuatorbridge.SetLogger(_parent._logger);

{region "Vertical : ActuatorDigitalBiLsPlusMinus"}
  Vertical.SetLogger(_parent._logger);
  Vertical.SetName(name:='Vertical', movePlusName:='Auf', moveMinusName:='Zu', plusName:='Offen', minusName:='Geschlossen');
  Vertical.SetSimulation(SEL(_parent._data.Config.Simulated, ActuatorDigitalSimulation.Disabled, ZEquipment.ActuatorDigitalSimulation.Automatic));
  Vertical.SetSimulationUncertainty(uncertainty:=10);
  Vertical.SetDelay(plusStartDuration:=0, plusEndDuration:=0, minusStartDuration:=0, minusEndDuration:=0, stop:=0);
  Vertical.SetSwitchDuration(plusDuration:=0.2, minusDuration:=0.2);
  Vertical.SetMovementDuration(plusDuration:=3, minusDuration:=3);
  Vertical.SetTimeout(plusDuration:=5, minusDuration:=5);
  _actuatorbridge.AddActuatorDigital(Vertical, publish := _parent._com.Publish.Equipment.Vertical, subscribe := _parent._com.Subscribe.Equipment.Vertical);
  _iobridge.AddDigitalOutput(Vertical.MinusOutput, publish := _parent._com.Publish.Equipment.VerticalZu, subscribe := _parent._com.Subscribe.Equipment.VerticalZu);
  _iobridge.AddDigitalOutput(Vertical.PlusOutput, publish := _parent._com.Publish.Equipment.VerticalAuf, subscribe := _parent._com.Subscribe.Equipment.VerticalAuf);
  _iobridge.AddDigitalInput(Vertical.MinusInput, publish := _parent._com.Publish.Equipment.VerticalGeschlossen, subscribe := _parent._com.Subscribe.Equipment.VerticalGeschlossen);
  _iobridge.AddDigitalInput(Vertical.PlusInput, publish := _parent._com.Publish.Equipment.VerticalOffen, subscribe := _parent._com.Subscribe.Equipment.VerticalOffen);
  {region "UserInitCode"}
  // put your individual init code for this Actuator here
  {endregion}

  {attribute 'ZId' := '6edc2aeb-8e0c-4ef7-9533-2d3679311649'}
{endregion}

{attribute '__ZwPlcUnitEquipmentImplementation__'} // Do not remove this attribute! It is used for code generation.

_isInitialized := TRUE;

END_FUNCTION_BLOCK

// ---- ZApp/Unit/Drilling/_Equipment/DrillingActuatorVertical.TcPOU
FUNCTION_BLOCK DrillingActuatorVertical EXTENDS ZEquipment.ActuatorDigitalBiLsPlusMinus

METHOD PUBLIC AufAsync
VAR_INPUT
  startToken : ZCore.IStartToken;
END_VAR
MovePlusAsync(startToken:=startToken);
END_METHOD

METHOD PUBLIC Geschlossen : BOOL
VAR_INPUT
END_VAR
Geschlossen := IsAtMinus();
END_METHOD

METHOD PUBLIC Offen : BOOL
VAR_INPUT
END_VAR
Offen := IsAtPlus();
END_METHOD

METHOD PUBLIC ZuAsync
VAR_INPUT
  startToken : ZCore.IStartToken;
END_VAR
MoveMinusAsync(startToken:=startToken);
END_METHOD

END_FUNCTION_BLOCK

// ---- ZApp/Unit/Drilling/_Equipment/DrillingAxis.TcPOU
/// This function block is a container for all axis objects that are used by this unit.
/// The parent of all objects can be directly transfered in their constructor (this is only relevant for equipment objects
/// that have to be managed (e.g. [DebouncedInput](xref:ZEquipment.DebouncedInput), [Light](xref:ZEquipment.Light), ...).
FUNCTION_BLOCK DrillingAxis EXTENDS DrillingContainer
VAR
  {attribute 'hide'}
  _axisbridge : ZApplication.AxisBridge(_parent);
END_VAR
VAR_INPUT

{attribute '__ZwPlcUnitEquipmentDeclaration__'} // Do not remove this attribute! It is used for code generation.
END_VAR

IF _isInitialized
THEN
  RETURN;
END_IF

  _axisbridge.SetLogger(_parent._logger);

{attribute '__ZwPlcUnitEquipmentImplementation__'} // Do not remove this attribute! It is used for code generation.

_isInitialized := TRUE;

END_FUNCTION_BLOCK

// ---- ZApp/Unit/Drilling/_Equipment/DrillingFieldbus.TcPOU
/// This function block is a container for all axis objects that are used by this unit.
/// The parent of all objects can be directly transfered in their constructor (this is only relevant for equipment objects
/// that have to be managed (e.g. [DebouncedInput](xref:ZEquipment.DebouncedInput), [Light](xref:ZEquipment.Light), ...).
FUNCTION_BLOCK DrillingFieldbus EXTENDS DrillingContainer
VAR
END_VAR
VAR_INPUT

{attribute '__ZwPlcUnitEquipmentDeclaration__'} // Do not remove this attribute! It is used for code generation.
END_VAR

IF _isInitialized
THEN
  RETURN;
END_IF

{attribute '__ZwPlcUnitEquipmentImplementation__'} // Do not remove this attribute! It is used for code generation.

_isInitialized := TRUE;

END_FUNCTION_BLOCK

// ---- ZApp/Unit/Drilling/_Equipment/DrillingLinkedUnit.TcPOU
/// This function block is a container for all linked units that are used by this unit.
/// Linked units can be addressed through their individual interface.
FUNCTION_BLOCK DrillingLinkedUnit EXTENDS DrillingContainer
VAR_INPUT

{attribute '__ZwPlcUnitEquipmentDeclaration__'} // Do not remove this attribute! It is used for code generation.
END_VAR

IF _isInitialized
THEN
  RETURN;
END_IF

{attribute '__ZwPlcUnitEquipmentImplementation__'} // Do not remove this attribute! It is used for code generation.

_isInitialized := TRUE;

END_FUNCTION_BLOCK

// ---- ZApp/Unit/Drilling/_States/DrillingSequenceBoot.TcPOU
FUNCTION_BLOCK DrillingSequenceBoot EXTENDS DrillingSequence IMPLEMENTS ZCore.ISequence
VAR
  _step : ZCore.Step(DrillingStep.BootBegin, DrillingStep.BootEnd);
END_VAR

IF OnStart(_step) THEN
  ; // init custom sequence variables here ...
END_IF

REPEAT
  LogStep();

  CASE _step.Index OF
    (* -------------------------------------------------------------------------------------------------------------------------------- *)
    DrillingStep.BootBegin:
    (* -------------------------------------------------------------------------------------------------------------------------------- *)
      IF _step.OnEntry()
      THEN
        // initialize equipment
        _io();
        _actuator();
        _fieldbus();
        _axis();
        _unit();
      END_IF
      
      _parent._objectManager.Cyclic();      
      Assert(_parent._objectManager);
      IF _parent._objectManager.Done
      THEN
        _step.SetNext(DrillingStep.BootEnd);
      END_IF

    (* -------------------------------------------------------------------------------------------------------------------------------- *)
    DrillingStep.BootEnd:
    (* -------------------------------------------------------------------------------------------------------------------------------- *)
      SetBusy(FALSE);
      
  ELSE
    Abort('sequence contains unhandled step');
  END_CASE
UNTIL _step.IsNotRepeatable() OR_ELSE NOT Busy END_REPEAT

END_FUNCTION_BLOCK

// ---- ZApp/Unit/Drilling/_SubObjects/DrillingSequence.TcPOU
FUNCTION_BLOCK DrillingSequence EXTENDS ZApplication.Sequence
VAR
  {attribute 'hide'}
  _parent : REFERENCE TO DrillingUnit;
  _io : REFERENCE TO DrillingIo;
  _actuator : REFERENCE TO DrillingActuator;
  _fieldbus : REFERENCE TO DrillingFieldbus;
  _axis : REFERENCE TO DrillingAxis;
  _data : REFERENCE TO DrillingDataRef;
  _unit : REFERENCE TO DrillingLinkedUnit;  
END_VAR

METHOD FB_init : BOOL
VAR_INPUT
  bInitRetains : BOOL; // if TRUE, the retain variables are initialized (warm start / cold start)
  bInCopyCode : BOOL;  // if TRUE, the instance afterwards gets moved into the copy code (online change)
  unit : REFERENCE TO DrillingUnit;
END_VAR
_parent REF= unit;
_alarming := unit._alarming;
_io REF= unit._equipment.Io;
_actuator REF= unit._equipment.Actuator;
_fieldbus REF= unit._equipment.Fieldbus;
_axis REF= unit._equipment.Axis;
_unit REF= unit._equipment.Unit;
_data REF= unit._data;
_loggerDiagnostics.SetLogger(unit._logger);
END_METHOD

